LIN {X 0,Y 168.479,Z 365.357,A -85,B 0,C 180,E1 -26143.185,E2 -26143.185} C_VEL
LIN {X 0,Y 172.542,Z 376.389,A -85,B 0,C 180,E1 -26145.975,E2 -26145.975} C_VEL
LIN {X 0,Y 176.909,Z 386.851,A -85,B 0,C 180,E1 -26149.006,E2 -26149.006} C_VEL
LIN {X 0,Y 181.024,Z 395.329,A -85,B 0,C 180,E1 -26151.737,E2 -26151.737} C_VEL
LIN {X 0,Y 187.387,Z 405.901,A -85,B 0,C 180,E1 -26155.598,E2 -26155.598} C_VEL
LIN {X 0,Y 193.546,Z 414.105,A -85,B 0,C 180,E1 -26158.901,E2 -26158.901} C_VEL
LIN {X 0,Y 201.697,Z 422.811,A -85,B 0,C 180,E1 -26162.738,E2 -26162.738} C_VEL
LIN {X 0,Y 211.071,Z 430.45,A -85,B 0,C 180,E1 -26166.449,E2 -26166.449} C_VEL
LIN {X 0,Y 223.559,Z 438.19,A -85,B 0,C 180,E1 -26170.576,E2 -26170.576} C_VEL
LIN {X 0,Y 237.874,Z 444.989,A -85,B 0,C 180,E1 -26174.579,E2 -26174.579} C_VEL
LIN {X 0,Y 246.269,Z 448.506,A -85,B 0,C 180,E1 -26176.803,E2 -26176.803} C_VEL
LIN {X 0,Y 253.879,Z 451.483,A -85,B 0,C 180,E1 -26178.827,E2 -26178.827} C_VEL
LIN {X 0,Y 260.174,Z 454.048,A -85,B 0,C 180,E1 -26180.673,E2 -26180.673} C_VEL
LIN {X 0,Y 265.402,Z 456.155,A -85,B 0,C 180,E1 -26182.392,E2 -26182.392} C_VEL
LIN {X 0,Y 269.49,Z 457.837,A -85,B 0,C 180,E1 -26184.012,E2 -26184.012} C_VEL
LIN {X 0,Y 272.317,Z 459.137,A -85,B 0,C 180,E1 -26185.559,E2 -26185.559} C_VEL
LIN {X 0,Y 274.967,Z 460.059,A -85,B 0,C 180,E1 -26187.07,E2 -26187.07} C_VEL
LIN {X 0,Y 276.58,Z 460.609,A -85,B 0,C 180,E1 -26188.544,E2 -26188.544} C_VEL
LIN {X 0,Y 277.495,Z 460.786,A -85,B 0,C 180,E1 -26190,E2 -26190} C_VEL
LIN {X 0,Y 276.59,Z 460.609,A -85,B 0,C 180,E1 -26191.456,E2 -26191.456} C_VEL
LIN {X 0,Y 274.514,Z 459.922,A -85,B 0,C 180,E1 -26193.194,E2 -26193.194} C_VEL
LIN {X 0,Y 272.314,Z 459.137,A -85,B 0,C 180,E1 -26194.441,E2 -26194.441} C_VEL
LIN {X 0,Y 268.697,Z 457.523,A -85,B 0,C 180,E1 -26196.329,E2 -26196.329} C_VEL
LIN {X 0,Y 265.405,Z 456.155,A -85,B 0,C 180,E1 -26197.608,E2 -26197.608} C_VEL
LIN {X 0,Y 260.168,Z 454.048,A -85,B 0,C 180,E1 -26199.328,E2 -26199.328} C_VEL
LIN {X 0,Y 251.344,Z 450.491,A -85,B 0,C 180,E1 -26201.863,E2 -26201.863} C_VEL
LIN {X 0,Y 239.95,Z 445.859,A -85,B 0,C 180,E1 -26204.865,E2 -26204.865} C_VEL
LIN {X 0,Y 226.946,Z 439.906,A -85,B 0,C 180,E1 -26208.442,E2 -26208.442} C_VEL
LIN {X 0,Y 213.379,Z 432.019,A -85,B 0,C 180,E1 -26212.749,E2 -26212.749} C_VEL
LIN {X 0,Y 202.838,Z 423.881,A -85,B 0,C 180,E1 -26216.771,E2 -26216.771} C_VEL
LIN {X 0,Y 195.211,Z 416.062,A -85,B 0,C 180,E1 -26220.267,E2 -26220.267} C_VEL
LIN {X 0,Y 188.321,Z 407.27,A -85,B 0,C 180,E1 -26223.869,E2 -26223.869} C_VEL
LIN {X 0,Y 182.818,Z 398.65,A -85,B 0,C 180,E1 -26227.094,E2 -26227.094} C_VEL
LIN {X 0,Y 178.539,Z 390.449,A -85,B 0,C 180,E1 -26229.863,E2 -26229.863} C_VEL
LIN {X 0,Y 174.431,Z 381.231,A -85,B 0,C 180,E1 -26232.669,E2 -26232.669} C_VEL
LIN {X 0,Y 170.461,Z 371.172,A -85,B 0,C 180,E1 -26235.399,E2 -26235.399} C_VEL
LIN {X 0,Y 166.541,Z 359.972,A -85,B 0,C 180,E1 -26238.043,E2 -26238.043} C_VEL
LIN {X 0,Y 161.005,Z 344.099,A -85,B 0,C 180,E1 -26241.47,E2 -26241.47} C_VEL
LIN {X 0,Y 157.401,Z 335.249,A -85,B 0,C 180,E1 -26243.828,E2 -26243.828} C_VEL
LIN {X 0,Y 153.095,Z 326.286,A -85,B 0,C 180,E1 -26246.861,E2 -26246.861} C_VEL
LIN {X 0,Y 148.607,Z 318.02,A -85,B 0,C 180,E1 -26250.423,E2 -26250.423} C_VEL
LIN {X 0,Y 144.236,Z 310.858,A -85,B 0,C 180,E1 -26254.476,E2 -26254.476} C_VEL
LIN {X 0,Y 141.455,Z 306.781,A -85,B 0,C 180,E1 -26257.5,E2 -26257.5} C_VEL
LIN {X 0,Y 138.818,Z 302.887,A -85,B 0,C 180,E1 -26260.923,E2 -26260.923} C_VEL
LIN {X 0,Y 136.47,Z 299.576,A -85,B 0,C 180,E1 -26264.698,E2 -26264.698} C_VEL
LIN {X 0,Y 135.748,Z 298.305,A -85,B 0,C 180,E1 -26266.148,E2 -26266.148} C_VEL
LIN {X 0,Y 133.362,Z 295.448,A -85,B 0,C 180,E1 -26272.431,E2 -26272.431} C_VEL
LIN {X 0,Y 132.753,Z 293.551,A -85,B 0,C 180,E1 -26276.207,E2 -26276.207} C_VEL
LIN {X 0,Y 132.567,Z 292.935,A -85,B 0,C 180,E1 -26280.002,E2 -26280.002} C_VEL
LIN {X 0,Y 132.838,Z 293.86,A -85,B 0,C 180,E1 -26284.173,E2 -26284.173} C_VEL
LIN {X 0,Y 135.419,Z 298.099,A -85,B 0,C 180,E1 -26292.839,E2 -26292.839} C_VEL
LIN {X 0,Y 136.074,Z 298.699,A -85,B 0,C 180,E1 -26294.108,E2 -26294.108} C_VEL
LIN {X 0,Y 138.286,Z 302.315,A -85,B 0,C 180,E1 -26297.947,E2 -26297.947} C_VEL
LIN {X 0,Y 139.47,Z 303.8,A -85,B 0,C 180,E1 -26299.599,E2 -26299.599} C_VEL
LIN {X 0,Y 142.595,Z 308.443,A -85,B 0,C 180,E1 -26303.416,E2 -26303.416} C_VEL
LIN {X 0,Y 145.282,Z 312.654,A -85,B 0,C 180,E1 -26306.196,E2 -26306.196} C_VEL
LIN {X 0,Y 147.772,Z 316.823,A -85,B 0,C 180,E1 -26308.497,E2 -26308.497} C_VEL
LIN {X 0,Y 151.056,Z 324.304,A -85,B 0,C 180,E1 -26311.368,E2 -26311.368} C_VEL
LIN {X 0,Y 155.191,Z 335.226,A -85,B 0,C 180,E1 -26314.649,E2 -26314.649} C_VEL
LIN {X 0,Y 156.553,Z 339.736,A -85,B 0,C 180,E1 -26315.706,E2 -26315.706} C_VEL
LIN {X 0,Y 154.15,Z 367.569,A -85,B 0,C 180,E1 -26316.786,E2 -26316.786} C_VEL
LIN {X 0,Y 152.045,Z 380.407,A -85,B 0,C 180,E1 -26317.581,E2 -26317.581} C_VEL
LIN {X 0,Y 148.731,Z 393.184,A -85,B 0,C 180,E1 -26318.77,E2 -26318.77} C_VEL
LIN {X 0,Y 145.566,Z 402.693,A -85,B 0,C 180,E1 -26319.964,E2 -26319.964} C_VEL
LIN {X 0,Y 141.889,Z 411.963,A -85,B 0,C 180,E1 -26321.482,E2 -26321.482} C_VEL
LIN {X 0,Y 137.794,Z 420.904,A -85,B 0,C 180,E1 -26323.381,E2 -26323.381} C_VEL
LIN {X 0,Y 133.305,Z 429.426,A -85,B 0,C 180,E1 -26325.689,E2 -26325.689} C_VEL
LIN {X 0,Y 129.058,Z 436.64,A -85,B 0,C 180,E1 -26328.158,E2 -26328.158} C_VEL
LIN {X 0,Y 125.1,Z 442.839,A -85,B 0,C 180,E1 -26330.802,E2 -26330.802} C_VEL
LIN {X 0,Y 120.656,Z 449.376,A -85,B 0,C 180,E1 -26334.375,E2 -26334.375} C_VEL
LIN {X 0,Y 115.978,Z 455.795,A -85,B 0,C 180,E1 -26338.997,E2 -26338.997} C_VEL
LIN {X 0,Y 111.963,Z 460.925,A -85,B 0,C 180,E1 -26343.935,E2 -26343.935} C_VEL
LIN {X 0,Y 108.804,Z 464.915,A -85,B 0,C 180,E1 -26349.191,E2 -26349.191} C_VEL
LIN {X 0,Y 106.703,Z 467.874,A -85,B 0,C 180,E1 -26354.725,E2 -26354.725} C_VEL
LIN {X 0,Y 105.26,Z 470.336,A -85,B 0,C 180,E1 -26362.326,E2 -26362.326} C_VEL
LIN {X 0,Y 105.047,Z 470.932,A -85,B 0,C 180,E1 -26366.164,E2 -26366.164} C_VEL
LIN {X 0,Y 105.171,Z 471.094,A -85,B 0,C 180,E1 -26370,E2 -26370} C_VEL
LIN {X 0,Y 105.037,Z 470.932,A -85,B 0,C 180,E1 -26373.836,E2 -26373.836} C_VEL
LIN {X 0,Y 105.221,Z 470.335,A -85,B 0,C 180,E1 -26377.677,E2 -26377.677} C_VEL
LIN {X 0,Y 106.666,Z 467.873,A -85,B 0,C 180,E1 -26385.281,E2 -26385.281} C_VEL
LIN {X 0,Y 108.804,Z 464.915,A -85,B 0,C 180,E1 -26390.809,E2 -26390.809} C_VEL
LIN {X 0,Y 111.962,Z 460.925,A -85,B 0,C 180,E1 -26396.065,E2 -26396.065} C_VEL
LIN {X 0,Y 115.965,Z 455.795,A -85,B 0,C 180,E1 -26401.007,E2 -26401.007} C_VEL
LIN {X 0,Y 120.653,Z 449.376,A -85,B 0,C 180,E1 -26405.626,E2 -26405.626} C_VEL
LIN {X 0,Y 126.045,Z 441.455,A -85,B 0,C 180,E1 -26409.882,E2 -26409.882} C_VEL
LIN {X 0,Y 131.144,Z 433.262,A -85,B 0,C 180,E1 -26413.099,E2 -26413.099} C_VEL
LIN {X 0,Y 136.077,Z 424.305,A -85,B 0,C 180,E1 -26415.775,E2 -26415.775} C_VEL
LIN {X 0,Y 140.078,Z 416.014,A -85,B 0,C 180,E1 -26417.734,E2 -26417.734} C_VEL
LIN {X 0,Y 144.316,Z 405.955,A -85,B 0,C 180,E1 -26419.545,E2 -26419.545} C_VEL
LIN {X 0,Y 147.754,Z 396.202,A -85,B 0,C 180,E1 -26420.887,E2 -26420.887} C_VEL
LIN {X 0,Y 150.623,Z 386.126,A -85,B 0,C 180,E1 -26421.941,E2 -26421.941} C_VEL
LIN {X 0,Y 152.867,Z 375.717,A -85,B 0,C 180,E1 -26422.747,E2 -26422.747} C_VEL
LIN {X 0,Y 154.387,Z 365.529,A -85,B 0,C 180,E1 -26423.295,E2 -26423.295} C_VEL
LIN {X 0,Y 156.505,Z 339.441,A -85,B 0,C 180,E1 -26424.342,E2 -26424.342} C_VEL
LIN {X 0,Y 153.574,Z 330.813,A -85,B 0,C 180,E1 -26426.591,E2 -26426.591} C_VEL
LIN {X 0,Y 149.887,Z 321.54,A -85,B 0,C 180,E1 -26429.621,E2 -26429.621} C_VEL
LIN {X 0,Y 147.162,Z 315.702,A -85,B 0,C 180,E1 -26432.054,E2 -26432.054} C_VEL
LIN {X 0,Y 143.791,Z 310.303,A -85,B 0,C 180,E1 -26435.3,E2 -26435.3} C_VEL
LIN {X 0,Y 141.753,Z 307.117,A -85,B 0,C 180,E1 -26437.547,E2 -26437.547} C_VEL
LIN {X 0,Y 140.373,Z 306.364,A -85,B 0,C 180,E1 -26439.042,E2 -26439.042} C_VEL
LIN {X 0,Y 135.987,Z 307.211,A -85,B 0,C 180,E1 -26444.335,E2 -26444.335} C_VEL
LIN {X 0,Y 135.091,Z 306.305,A -85,B 0,C 180,E1 -26445.924,E2 -26445.924} C_VEL
LIN {X 0,Y 134.567,Z 305.22,A -85,B 0,C 180,E1 -26447.078,E2 -26447.078} C_VEL
LIN {X 0,Y 132.204,Z 301.989,A -85,B 0,C 180,E1 -26454.087,E2 -26454.087} C_VEL
LIN {X 0,Y 131.781,Z 300.34,A -85,B 0,C 180,E1 -26457.706,E2 -26457.706} C_VEL
LIN {X 0,Y 131.702,Z 299.984,A -85,B 0,C 180,E1 -26459.998,E2 -26459.998} C_VEL
LIN {X 0,Y 131.918,Z 300.847,A -85,B 0,C 180,E1 -26464.199,E2 -26464.199} C_VEL
LIN {X 0,Y 134.157,Z 304.913,A -85,B 0,C 180,E1 -26472.454,E2 -26472.454} C_VEL
LIN {X 0,Y 134.778,Z 305.568,A -85,B 0,C 180,E1 -26473.762,E2 -26473.762} C_VEL
LIN {X 0,Y 137.237,Z 309.489,A -85,B 0,C 180,E1 -26478.173,E2 -26478.173} C_VEL
LIN {X 0,Y 140.562,Z 314.653,A -85,B 0,C 180,E1 -26482.651,E2 -26482.651} C_VEL
LIN {X 0,Y 143.908,Z 320.11,A -85,B 0,C 180,E1 -26486.294,E2 -26486.294} C_VEL
LIN {X 0,Y 147.845,Z 327.198,A -85,B 0,C 180,E1 -26489.941,E2 -26489.941} C_VEL
LIN {X 0,Y 152.298,Z 336.274,A -85,B 0,C 180,E1 -26493.523,E2 -26493.523} C_VEL
LIN {X 0,Y 156.232,Z 345.744,A -85,B 0,C 180,E1 -26496.385,E2 -26496.385} C_VEL
LIN {X 0,Y 160.334,Z 358.02,A -85,B 0,C 180,E1 -26499.258,E2 -26499.258} C_VEL
LIN {X 0,Y 163.619,Z 368.614,A -85,B 0,C 180,E1 -26501.74,E2 -26501.74} C_VEL
LIN {X 0,Y 166.649,Z 377.879,A -85,B 0,C 180,E1 -26504.198,E2 -26504.198} C_VEL
LIN {X 0,Y 169.964,Z 386.802,A -85,B 0,C 180,E1 -26506.88,E2 -26506.88} C_VEL
LIN {X 0,Y 174.041,Z 396.438,A -85,B 0,C 180,E1 -26510.105,E2 -26510.105} C_VEL
LIN {X 0,Y 178.97,Z 405.713,A -85,B 0,C 180,E1 -26513.612,E2 -26513.612} C_VEL
LIN {X 0,Y 184.343,Z 413.859,A -85,B 0,C 180,E1 -26517.005,E2 -26517.005} C_VEL
LIN {X 0,Y 190.846,Z 421.669,A -85,B 0,C 180,E1 -26520.576,E2 -26520.576} C_VEL
LIN {X 0,Y 198.48,Z 428.958,A -85,B 0,C 180,E1 -26524.202,E2 -26524.202} C_VEL
LIN {X 0,Y 208.831,Z 436.357,A -85,B 0,C 180,E1 -26528.273,E2 -26528.273} C_VEL
LIN {X 0,Y 221.286,Z 443.055,A -85,B 0,C 180,E1 -26532.321,E2 -26532.321} C_VEL
LIN {X 0,Y 235.113,Z 448.819,A -85,B 0,C 180,E1 -26536.165,E2 -26536.165} C_VEL
LIN {X 0,Y 246.762,Z 453.049,A -85,B 0,C 180,E1 -26539.287,E2 -26539.287} C_VEL
LIN {X 0,Y 250.341,Z 454.315,A -85,B 0,C 180,E1 -26540.303,E2 -26540.303} C_VEL
LIN {X 0,Y 256.375,Z 456.402,A -85,B 0,C 180,E1 -26542.122,E2 -26542.122} C_VEL
LIN {X 0,Y 261.472,Z 458.211,A -85,B 0,C 180,E1 -26543.983,E2 -26543.983} C_VEL
LIN {X 0,Y 264.47,Z 459.349,A -85,B 0,C 180,E1 -26545.427,E2 -26545.427} C_VEL
LIN {X 0,Y 267.409,Z 460.312,A -85,B 0,C 180,E1 -26547.069,E2 -26547.069} C_VEL
LIN {X 0,Y 269.257,Z 460.807,A -85,B 0,C 180,E1 -26548.504,E2 -26548.504} C_VEL
LIN {X 0,Y 270.327,Z 460.977,A -85,B 0,C 180,E1 -26550,E2 -26550} C_VEL
LIN {X 0,Y 269.264,Z 460.807,A -85,B 0,C 180,E1 -26551.496,E2 -26551.496} C_VEL
LIN {X 0,Y 267.259,Z 460.27,A -85,B 0,C 180,E1 -26553.015,E2 -26553.015} C_VEL
LIN {X 0,Y 264.443,Z 459.349,A -85,B 0,C 180,E1 -26554.573,E2 -26554.573} C_VEL
LIN {X 0,Y 261.037,Z 458.069,A -85,B 0,C 180,E1 -26556.182,E2 -26556.182} C_VEL
LIN {X 0,Y 255.572,Z 456.138,A -85,B 0,C 180,E1 -26558.13,E2 -26558.13} C_VEL
LIN {X 0,Y 249.683,Z 454.083,A -85,B 0,C 180,E1 -26559.886,E2 -26559.886} C_VEL
LIN {X 0,Y 243.138,Z 451.778,A -85,B 0,C 180,E1 -26561.674,E2 -26561.674} C_VEL
LIN {X 0,Y 232.36,Z 447.741,A -85,B 0,C 180,E1 -26564.566,E2 -26564.566} C_VEL
LIN {X 0,Y 221.299,Z 443.027,A -85,B 0,C 180,E1 -26567.689,E2 -26567.689} C_VEL
LIN {X 0,Y 208.858,Z 436.356,A -85,B 0,C 180,E1 -26571.725,E2 -26571.725} C_VEL
LIN {X 0,Y 200.699,Z 430.75,A -85,B 0,C 180,E1 -26574.848,E2 -26574.848} C_VEL
LIN {X 0,Y 193.245,Z 424.166,A -85,B 0,C 180,E1 -26578.215,E2 -26578.215} C_VEL
LIN {X 0,Y 186.275,Z 416.336,A -85,B 0,C 180,E1 -26581.884,E2 -26581.884} C_VEL
LIN {X 0,Y 180.695,Z 408.562,A -85,B 0,C 180,E1 -26585.239,E2 -26585.239} C_VEL
LIN {X 0,Y 175.593,Z 399.762,A -85,B 0,C 180,E1 -26588.698,E2 -26588.698} C_VEL
LIN {X 0,Y 171.748,Z 391.161,A -85,B 0,C 180,E1 -26591.687,E2 -26591.687} C_VEL
LIN {X 0,Y 168.397,Z 382.706,A -85,B 0,C 180,E1 -26594.384,E2 -26594.384} C_VEL
LIN {X 0,Y 164.92,Z 372.651,A -85,B 0,C 180,E1 -26597.223,E2 -26597.223} C_VEL
LIN {X 0,Y 161.358,Z 361.267,A -85,B 0,C 180,E1 -26600.028,E2 -26600.028} C_VEL
LIN {X 0,Y 157.135,Z 348.285,A -85,B 0,C 180,E1 -26602.977,E2 -26602.977} C_VEL
LIN {X 0,Y 153.766,Z 339.696,A -85,B 0,C 180,E1 -26605.376,E2 -26605.376} C_VEL
LIN {X 0,Y 149.798,Z 331.089,A -85,B 0,C 180,E1 -26608.425,E2 -26608.425} C_VEL
LIN {X 0,Y 145.89,Z 323.573,A -85,B 0,C 180,E1 -26611.802,E2 -26611.802} C_VEL
LIN {X 0,Y 141.921,Z 316.824,A -85,B 0,C 180,E1 -26615.791,E2 -26615.791} C_VEL
LIN {X 0,Y 139.553,Z 313.107,A -85,B 0,C 180,E1 -26618.587,E2 -26618.587} C_VEL
LIN {X 0,Y 137.239,Z 309.488,A -85,B 0,C 180,E1 -26621.826,E2 -26621.826} C_VEL
LIN {X 0,Y 134.859,Z 305.757,A -85,B 0,C 180,E1 -26626.055,E2 -26626.055} C_VEL
LIN {X 0,Y 134.162,Z 304.871,A -85,B 0,C 180,E1 -26627.546,E2 -26627.546} C_VEL
LIN {X 0,Y 132.174,Z 301.855,A -85,B 0,C 180,E1 -26633.897,E2 -26633.897} C_VEL
LIN {X 0,Y 131.811,Z 300.43,A -85,B 0,C 180,E1 -26636.945,E2 -26636.945} C_VEL
LIN {X 0,Y 131.707,Z 300.081,A -85,B 0,C 180,E1 -26640.766,E2 -26640.766} C_VEL
LIN {X 0,Y 131.925,Z 300.918,A -85,B 0,C 180,E1 -26643.915,E2 -26643.915} C_VEL
LIN {X 0,Y 134.298,Z 305.023,A -85,B 0,C 180,E1 -26652.372,E2 -26652.372} C_VEL
LIN {X 0,Y 134.859,Z 305.768,A -85,B 0,C 180,E1 -26653.565,E2 -26653.565} C_VEL
LIN {X 0,Y 137.95,Z 310.612,A -85,B 0,C 180,E1 -26658.858,E2 -26658.858} C_VEL
LIN {X 0,Y 140.594,Z 314.65,A -85,B 0,C 180,E1 -26662.3,E2 -26662.3} C_VEL
LIN {X 0,Y 144.211,Z 320.604,A -85,B 0,C 180,E1 -26666.211,E2 -26666.211} C_VEL
LIN {X 0,Y 146.759,Z 326.225,A -85,B 0,C 180,E1 -26668.712,E2 -26668.712} C_VEL
LIN {X 0,Y 150.274,Z 335.658,A -85,B 0,C 180,E1 -26671.894,E2 -26671.894} C_VEL
LIN {X 0,Y 152.306,Z 342.009,A -85,B 0,C 180,E1 -26673.625,E2 -26673.625} C_VEL
LIN {X 0,Y 150.039,Z 367.082,A -85,B 0,C 180,E1 -26674.597,E2 -26674.597} C_VEL
LIN {X 0,Y 147.79,Z 380.354,A -85,B 0,C 180,E1 -26675.408,E2 -26675.408} C_VEL
LIN {X 0,Y 144.398,Z 392.992,A -85,B 0,C 180,E1 -26676.576,E2 -26676.576} C_VEL
LIN {X 0,Y 141.112,Z 402.501,A -85,B 0,C 180,E1 -26677.755,E2 -26677.755} C_VEL
LIN {X 0,Y 137.277,Z 411.77,A -85,B 0,C 180,E1 -26679.256,E2 -26679.256} C_VEL
LIN {X 0,Y 133.008,Z 420.711,A -85,B 0,C 180,E1 -26681.153,E2 -26681.153} C_VEL
LIN {X 0,Y 128.322,Z 429.234,A -85,B 0,C 180,E1 -26683.475,E2 -26683.475} C_VEL
LIN {X 0,Y 123.832,Z 436.447,A -85,B 0,C 180,E1 -26685.954,E2 -26685.954} C_VEL
LIN {X 0,Y 119.662,Z 442.645,A -85,B 0,C 180,E1 -26688.644,E2 -26688.644} C_VEL
LIN {X 0,Y 114.934,Z 449.182,A -85,B 0,C 180,E1 -26692.304,E2 -26692.304} C_VEL
LIN {X 0,Y 111.518,Z 453.685,A -85,B 0,C 180,E1 -26695.446,E2 -26695.446} C_VEL
LIN {X 0,Y 106.899,Z 459.176,A -85,B 0,C 180,E1 -26700.457,E2 -26700.457} C_VEL
LIN {X 0,Y 103.208,Z 463.503,A -85,B 0,C 180,E1 -26705.885,E2 -26705.885} C_VEL
LIN {X 0,Y 101.256,Z 465.874,A -85,B 0,C 180,E1 -26709.694,E2 -26709.694} C_VEL
LIN {X 0,Y 99.828,Z 467.68,A -85,B 0,C 180,E1 -26713.644,E2 -26713.644} C_VEL
LIN {X 0,Y 98.209,Z 470.142,A -85,B 0,C 180,E1 -26721.771,E2 -26721.771} C_VEL
LIN {X 0,Y 97.952,Z 470.739,A -85,B 0,C 180,E1 -26725.886,E2 -26725.886} C_VEL
LIN {X 0,Y 98.077,Z 470.902,A -85,B 0,C 180,E1 -26730,E2 -26730} C_VEL
LIN {X 0,Y 97.943,Z 470.739,A -85,B 0,C 180,E1 -26734.115,E2 -26734.115} C_VEL
LIN {X 0,Y 98.178,Z 470.141,A -85,B 0,C 180,E1 -26738.231,E2 -26738.231} C_VEL
LIN {X 0,Y 99.798,Z 467.679,A -85,B 0,C 180,E1 -26746.361,E2 -26746.361} C_VEL
LIN {X 0,Y 102.181,Z 464.722,A -85,B 0,C 180,E1 -26752.228,E2 -26752.228} C_VEL
LIN {X 0,Y 105.595,Z 460.731,A -85,B 0,C 180,E1 -26757.768,E2 -26757.768} C_VEL
LIN {X 0,Y 109.929,Z 455.602,A -85,B 0,C 180,E1 -26762.917,E2 -26762.917} C_VEL
LIN {X 0,Y 114.092,Z 450.286,A -85,B 0,C 180,E1 -26766.962,E2 -26766.962} C_VEL
LIN {X 0,Y 118.658,Z 444.02,A -85,B 0,C 180,E1 -26770.656,E2 -26770.656} C_VEL
LIN {X 0,Y 122.787,Z 438.073,A -85,B 0,C 180,E1 -26773.381,E2 -26773.381} C_VEL
LIN {X 0,Y 127.157,Z 431.15,A -85,B 0,C 180,E1 -26775.931,E2 -26775.931} C_VEL
LIN {X 0,Y 131.807,Z 422.978,A -85,B 0,C 180,E1 -26778.287,E2 -26778.287} C_VEL
LIN {X 0,Y 136.035,Z 414.471,A -85,B 0,C 180,E1 -26780.218,E2 -26780.218} C_VEL
LIN {X 0,Y 139.808,Z 405.762,A -85,B 0,C 180,E1 -26781.762,E2 -26781.762} C_VEL
LIN {X 0,Y 143.391,Z 396.01,A -85,B 0,C 180,E1 -26783.084,E2 -26783.084} C_VEL
LIN {X 0,Y 146.359,Z 385.933,A -85,B 0,C 180,E1 -26784.127,E2 -26784.127} C_VEL
LIN {X 0,Y 148.53,Z 376.276,A -85,B 0,C 180,E1 -26784.879,E2 -26784.879} C_VEL
LIN {X 0,Y 150.171,Z 366.091,A -85,B 0,C 180,E1 -26785.427,E2 -26785.427} C_VEL
LIN {X 0,Y 152.308,Z 341.993,A -85,B 0,C 180,E1 -26786.376,E2 -26786.376} C_VEL
LIN {X 0,Y 149.957,Z 334.8,A -85,B 0,C 180,E1 -26788.376,E2 -26788.376} C_VEL
LIN {X 0,Y 146.839,Z 326.47,A -85,B 0,C 180,E1 -26791.208,E2 -26791.208} C_VEL
LIN {X 0,Y 144.294,Z 320.735,A -85,B 0,C 180,E1 -26793.708,E2 -26793.708} C_VEL
LIN {X 0,Y 140.107,Z 313.769,A -85,B 0,C 180,E1 -26798.304,E2 -26798.304} C_VEL
LIN {X 0,Y 137.065,Z 309.285,A -85,B 0,C 180,E1 -26802.466,E2 -26802.466} C_VEL
LIN {X 0,Y 135.091,Z 306.305,A -85,B 0,C 180,E1 -26805.924,E2 -26805.924} C_VEL
LIN {X 0,Y 134.359,Z 305.169,A -85,B 0,C 180,E1 -26807.476,E2 -26807.476} C_VEL
LIN {X 0,Y 133.244,Z 304.74,A -85,B 0,C 180,E1 -26809.939,E2 -26809.939} C_VEL
LIN {X 0,Y 131.692,Z 305.939,A -85,B 0,C 180,E1 -26814.187,E2 -26814.187} C_VEL
LIN {X 0,Y 130.877,Z 307.119,A -85,B 0,C 180,E1 -26818.579,E2 -26818.579} C_VEL
LIN {X 0,Y 130.838,Z 307.095,A -85,B 0,C 180,E1 -26819.468,E2 -26819.468} C_VEL
LIN {X 0,Y 130.969,Z 307.678,A -85,B 0,C 180,E1 -26823.459,E2 -26823.459} C_VEL
LIN {X 0,Y 132.983,Z 311.787,A -85,B 0,C 180,E1 -26831.824,E2 -26831.824} C_VEL
LIN {X 0,Y 133.57,Z 312.561,A -85,B 0,C 180,E1 -26833.171,E2 -26833.171} C_VEL
LIN {X 0,Y 136.341,Z 317.175,A -85,B 0,C 180,E1 -26838.297,E2 -26838.297} C_VEL
LIN {X 0,Y 138.859,Z 321.337,A -85,B 0,C 180,E1 -26841.823,E2 -26841.823} C_VEL
LIN {X 0,Y 141.692,Z 326.216,A -85,B 0,C 180,E1 -26845.13,E2 -26845.13} C_VEL
LIN {X 0,Y 145.284,Z 333.104,A -85,B 0,C 180,E1 -26848.727,E2 -26848.727} C_VEL
LIN {X 0,Y 149.381,Z 342.043,A -85,B 0,C 180,E1 -26852.296,E2 -26852.296} C_VEL
LIN {X 0,Y 152.673,Z 350.479,A -85,B 0,C 180,E1 -26854.903,E2 -26854.903} C_VEL
LIN {X 0,Y 156.081,Z 361.51,A -85,B 0,C 180,E1 -26857.638,E2 -26857.638} C_VEL
LIN {X 0,Y 158.454,Z 370.323,A -85,B 0,C 180,E1 -26859.816,E2 -26859.816} C_VEL
LIN {X 0,Y 160.646,Z 378.117,A -85,B 0,C 180,E1 -26861.951,E2 -26861.951} C_VEL
LIN {X 0,Y 163.869,Z 388.405,A -85,B 0,C 180,E1 -26865.151,E2 -26865.151} C_VEL
LIN {X 0,Y 167.12,Z 397.069,A -85,B 0,C 180,E1 -26868.19,E2 -26868.19} C_VEL
LIN {X 0,Y 170.834,Z 405.401,A -85,B 0,C 180,E1 -26871.409,E2 -26871.409} C_VEL
LIN {X 0,Y 176.395,Z 414.906,A -85,B 0,C 180,E1 -26875.559,E2 -26875.559} C_VEL
LIN {X 0,Y 181.738,Z 421.97,A -85,B 0,C 180,E1 -26878.951,E2 -26878.951} C_VEL
LIN {X 0,Y 189.22,Z 429.789,A -85,B 0,C 180,E1 -26883.048,E2 -26883.048} C_VEL
LIN {X 0,Y 198.337,Z 436.791,A -85,B 0,C 180,E1 -26887.114,E2 -26887.114} C_VEL
LIN {X 0,Y 208.358,Z 442.584,A -85,B 0,C 180,E1 -26890.809,E2 -26890.809} C_VEL
LIN {X 0,Y 219.136,Z 447.41,A -85,B 0,C 180,E1 -26894.18,E2 -26894.18} C_VEL
LIN {X 0,Y 232.085,Z 452.082,A -85,B 0,C 180,E1 -26897.762,E2 -26897.762} C_VEL
LIN {X 0,Y 242.26,Z 455.294,A -85,B 0,C 180,E1 -26900.514,E2 -26900.514} C_VEL
LIN {X 0,Y 248.225,Z 457.108,A -85,B 0,C 180,E1 -26902.28,E2 -26902.28} C_VEL
LIN {X 0,Y 254.243,Z 458.919,A -85,B 0,C 180,E1 -26904.339,E2 -26904.339} C_VEL
LIN {X 0,Y 256.387,Z 459.567,A -85,B 0,C 180,E1 -26905.283,E2 -26905.283} C_VEL
LIN {X 0,Y 260.309,Z 460.676,A -85,B 0,C 180,E1 -26907.354,E2 -26907.354} C_VEL
LIN {X 0,Y 261.833,Z 461.008,A -85,B 0,C 180,E1 -26908.462,E2 -26908.462} C_VEL
LIN {X 0,Y 263.136,Z 461.168,A -85,B 0,C 180,E1 -26910,E2 -26910} C_VEL
LIN {X 0,Y 261.838,Z 461.007,A -85,B 0,C 180,E1 -26911.538,E2 -26911.538} C_VEL
LIN {X 0,Y 259.49,Z 460.482,A -85,B 0,C 180,E1 -26913.105,E2 -26913.105} C_VEL
LIN {X 0,Y 256.372,Z 459.567,A -85,B 0,C 180,E1 -26914.717,E2 -26914.717} C_VEL
LIN {X 0,Y 254.243,Z 458.92,A -85,B 0,C 180,E1 -26915.66,E2 -26915.66} C_VEL
LIN {X 0,Y 248.225,Z 457.108,A -85,B 0,C 180,E1 -26917.72,E2 -26917.72} C_VEL
LIN {X 0,Y 239.922,Z 454.596,A -85,B 0,C 180,E1 -26920.123,E2 -26920.123} C_VEL
LIN {X 0,Y 230.494,Z 451.563,A -85,B 0,C 180,E1 -26922.658,E2 -26922.658} C_VEL
LIN {X 0,Y 219.14,Z 447.401,A -85,B 0,C 180,E1 -26925.824,E2 -26925.824} C_VEL
LIN {X 0,Y 206.255,Z 441.488,A -85,B 0,C 180,E1 -26929.922,E2 -26929.922} C_VEL
LIN {X 0,Y 196.267,Z 435.387,A -85,B 0,C 180,E1 -26933.748,E2 -26933.748} C_VEL
LIN {X 0,Y 187.142,Z 427.784,A -85,B 0,C 180,E1 -26938.054,E2 -26938.054} C_VEL
LIN {X 0,Y 179.291,Z 418.917,A -85,B 0,C 180,E1 -26942.57,E2 -26942.57} C_VEL
LIN {X 0,Y 173.202,Z 409.793,A -85,B 0,C 180,E1 -26946.74,E2 -26946.74} C_VEL
LIN {X 0,Y 169.134,Z 401.905,A -85,B 0,C 180,E1 -26950.007,E2 -26950.007} C_VEL
LIN {X 0,Y 165.129,Z 391.922,A -85,B 0,C 180,E1 -26953.655,E2 -26953.655} C_VEL
LIN {X 0,Y 162.036,Z 382.699,A -85,B 0,C 180,E1 -26956.674,E2 -26956.674} C_VEL
LIN {X 0,Y 158.946,Z 372.137,A -85,B 0,C 180,E1 -26959.712,E2 -26959.712} C_VEL
LIN {X 0,Y 155.937,Z 360.94,A -85,B 0,C 180,E1 -26962.525,E2 -26962.525} C_VEL
LIN {X 0,Y 152.677,Z 350.493,A -85,B 0,C 180,E1 -26965.094,E2 -26965.094} C_VEL
LIN {X 0,Y 149.475,Z 342.254,A -85,B 0,C 180,E1 -26967.628,E2 -26967.628} C_VEL
LIN {X 0,Y 145.285,Z 333.096,A -85,B 0,C 180,E1 -26971.273,E2 -26971.273} C_VEL
LIN {X 0,Y 141.69,Z 326.232,A -85,B 0,C 180,E1 -26974.87,E2 -26974.87} C_VEL
LIN {X 0,Y 139.196,Z 321.927,A -85,B 0,C 180,E1 -26977.75,E2 -26977.75} C_VEL
LIN {X 0,Y 137.53,Z 319.166,A -85,B 0,C 180,E1 -26979.944,E2 -26979.944} C_VEL
LIN {X 0,Y 135.568,Z 315.944,A -85,B 0,C 180,E1 -26982.95,E2 -26982.95} C_VEL
LIN {X 0,Y 133.307,Z 312.004,A -85,B 0,C 180,E1 -26987.465,E2 -26987.465} C_VEL
LIN {X 0,Y 131.241,Z 308.956,A -85,B 0,C 180,E1 -26994.143,E2 -26994.143} C_VEL
LIN {X 0,Y 130.94,Z 307.531,A -85,B 0,C 180,E1 -26996.925,E2 -26996.925} C_VEL
LIN {X 0,Y 130.842,Z 307.127,A -85,B 0,C 180,E1 -27000.771,E2 -27000.771} C_VEL
LIN {X 0,Y 131.049,Z 308.068,A -85,B 0,C 180,E1 -27003.942,E2 -27003.942} C_VEL
LIN {X 0,Y 133.112,Z 311.88,A -85,B 0,C 180,E1 -27011.732,E2 -27011.732} C_VEL
LIN {X 0,Y 133.622,Z 312.703,A -85,B 0,C 180,E1 -27012.918,E2 -27012.918} C_VEL
LIN {X 0,Y 136.289,Z 317.073,A -85,B 0,C 180,E1 -27017.831,E2 -27017.831} C_VEL
LIN {X 0,Y 138.782,Z 321.164,A -85,B 0,C 180,E1 -27021.337,E2 -27021.337} C_VEL
LIN {X 0,Y 141.981,Z 326.752,A -85,B 0,C 180,E1 -27025.06,E2 -27025.06} C_VEL
LIN {X 0,Y 144.559,Z 333.019,A -85,B 0,C 180,E1 -27027.804,E2 -27027.804} C_VEL
LIN {X 0,Y 148.18,Z 343.951,A -85,B 0,C 180,E1 -27031.34,E2 -27031.34} C_VEL
LIN {X 0,Y 148.118,Z 346.245,A -85,B 0,C 180,E1 -27031.508,E2 -27031.508} C_VEL
LIN {X 0,Y 146.034,Z 367.636,A -85,B 0,C 180,E1 -27032.343,E2 -27032.343} C_VEL
LIN {X 0,Y 143.414,Z 381.697,A -85,B 0,C 180,E1 -27033.22,E2 -27033.22} C_VEL
LIN {X 0,Y 140.285,Z 392.799,A -85,B 0,C 180,E1 -27034.248,E2 -27034.248} C_VEL
LIN {X 0,Y 136.878,Z 402.308,A -85,B 0,C 180,E1 -27035.403,E2 -27035.403} C_VEL
LIN {X 0,Y 132.907,Z 411.578,A -85,B 0,C 180,E1 -27036.89,E2 -27036.89} C_VEL
LIN {X 0,Y 128.432,Z 420.517,A -85,B 0,C 180,E1 -27038.76,E2 -27038.76} C_VEL
LIN {X 0,Y 123.546,Z 429.041,A -85,B 0,C 180,E1 -27041.085,E2 -27041.085} C_VEL
LIN {X 0,Y 118.817,Z 436.253,A -85,B 0,C 180,E1 -27043.566,E2 -27043.566} C_VEL
LIN {X 0,Y 114.399,Z 442.451,A -85,B 0,C 180,E1 -27046.28,E2 -27046.28} C_VEL
LIN {X 0,Y 109.365,Z 448.988,A -85,B 0,C 180,E1 -27050.013,E2 -27050.013} C_VEL
LIN {X 0,Y 104.016,Z 455.408,A -85,B 0,C 180,E1 -27054.948,E2 -27054.948} C_VEL
LIN {X 0,Y 99.324,Z 460.537,A -85,B 0,C 180,E1 -27060.31,E2 -27060.31} C_VEL
LIN {X 0,Y 95.608,Z 464.528,A -85,B 0,C 180,E1 -27066.153,E2 -27066.153} C_VEL
LIN {X 0,Y 93.003,Z 467.486,A -85,B 0,C 180,E1 -27072.406,E2 -27072.406} C_VEL
LIN {X 0,Y 91.164,Z 469.949,A -85,B 0,C 180,E1 -27081.131,E2 -27081.131} C_VEL
LIN {X 0,Y 90.88,Z 470.547,A -85,B 0,C 180,E1 -27085.565,E2 -27085.565} C_VEL
LIN {X 0,Y 90.976,Z 470.709,A -85,B 0,C 180,E1 -27090,E2 -27090} C_VEL
LIN {X 0,Y 90.873,Z 470.546,A -85,B 0,C 180,E1 -27094.436,E2 -27094.436} C_VEL
LIN {X 0,Y 91.138,Z 469.948,A -85,B 0,C 180,E1 -27098.872,E2 -27098.872} C_VEL
LIN {X 0,Y 92.979,Z 467.486,A -85,B 0,C 180,E1 -27107.599,E2 -27107.599} C_VEL
LIN {X 0,Y 95.608,Z 464.528,A -85,B 0,C 180,E1 -27113.847,E2 -27113.847} C_VEL
LIN {X 0,Y 99.322,Z 460.537,A -85,B 0,C 180,E1 -27119.69,E2 -27119.69} C_VEL
LIN {X 0,Y 104.008,Z 455.408,A -85,B 0,C 180,E1 -27125.055,E2 -27125.055} C_VEL
LIN {X 0,Y 109.36,Z 448.988,A -85,B 0,C 180,E1 -27129.989,E2 -27129.989} C_VEL
LIN {X 0,Y 115.494,Z 441.069,A -85,B 0,C 180,E1 -27134.41,E2 -27134.41} C_VEL
LIN {X 0,Y 121.144,Z 432.875,A -85,B 0,C 180,E1 -27137.703,E2 -27137.703} C_VEL
LIN {X 0,Y 126.576,Z 423.919,A -85,B 0,C 180,E1 -27140.389,E2 -27140.389} C_VEL
LIN {X 0,Y 130.951,Z 415.628,A -85,B 0,C 180,E1 -27142.336,E2 -27142.336} C_VEL
LIN {X 0,Y 135.533,Z 405.569,A -85,B 0,C 180,E1 -27144.118,E2 -27144.118} C_VEL
LIN {X 0,Y 139.25,Z 395.818,A -85,B 0,C 180,E1 -27145.416,E2 -27145.416} C_VEL
LIN {X 0,Y 142.316,Z 385.74,A -85,B 0,C 180,E1 -27146.443,E2 -27146.443} C_VEL
LIN {X 0,Y 144.682,Z 375.482,A -85,B 0,C 180,E1 -27147.218,E2 -27147.218} C_VEL
LIN {X 0,Y 146.319,Z 365.419,A -85,B 0,C 180,E1 -27147.738,E2 -27147.738} C_VEL
LIN {X 0,Y 148.264,Z 344.353,A -85,B 0,C 180,E1 -27148.571,E2 -27148.571} C_VEL
LIN {X 0,Y 146.173,Z 337.686,A -85,B 0,C 180,E1 -27150.571,E2 -27150.571} C_VEL
LIN {X 0,Y 143.3,Z 329.775,A -85,B 0,C 180,E1 -27153.511,E2 -27153.511} C_VEL
LIN {X 0,Y 141.519,Z 325.961,A -85,B 0,C 180,E1 -27155.433,E2 -27155.433} C_VEL
LIN {X 0,Y 138.134,Z 319.987,A -85,B 0,C 180,E1 -27159.524,E2 -27159.524} C_VEL
LIN {X 0,Y 135.513,Z 315.851,A -85,B 0,C 180,E1 -27163.425,E2 -27163.425} C_VEL
LIN {X 0,Y 133.311,Z 312.06,A -85,B 0,C 180,E1 -27167.825,E2 -27167.825} C_VEL
LIN {X 0,Y 131.121,Z 308.457,A -85,B 0,C 180,E1 -27175.387,E2 -27175.387} C_VEL
LIN {X 0,Y 130.868,Z 307.256,A -85,B 0,C 180,E1 -27178.46,E2 -27178.46} C_VEL
LIN {X 0,Y 130.838,Z 307.095,A -85,B 0,C 180,E1 -27179.468,E2 -27179.468} C_VEL
LIN {X 0,Y 130.817,Z 307.339,A -85,B 0,C 180,E1 -27181.17,E2 -27181.17} C_VEL
LIN {X 0,Y 130.84,Z 308.932,A -85,B 0,C 180,E1 -27183.647,E2 -27183.647} C_VEL
LIN {X 0,Y 130.964,Z 311.456,A -85,B 0,C 180,E1 -27185.994,E2 -27185.994} C_VEL
LIN {X 0,Y 131.373,Z 315.507,A -85,B 0,C 180,E1 -27189.08,E2 -27189.08} C_VEL
LIN {X 0,Y 132.245,Z 319.17,A -85,B 0,C 180,E1 -27192.212,E2 -27192.212} C_VEL
LIN {X 0,Y 134.676,Z 323.541,A -85,B 0,C 180,E1 -27197.166,E2 -27197.166} C_VEL
LIN {X 0,Y 137.086,Z 327.797,A -85,B 0,C 180,E1 -27200.832,E2 -27200.832} C_VEL
LIN {X 0,Y 139.853,Z 332.901,A -85,B 0,C 180,E1 -27204.294,E2 -27204.294} C_VEL
LIN {X 0,Y 143.216,Z 339.893,A -85,B 0,C 180,E1 -27207.892,E2 -27207.892} C_VEL
LIN {X 0,Y 146.733,Z 348.236,A -85,B 0,C 180,E1 -27211.19,E2 -27211.19} C_VEL
LIN {X 0,Y 149.632,Z 356.394,A -85,B 0,C 180,E1 -27213.696,E2 -27213.696} C_VEL
LIN {X 0,Y 152.716,Z 368.599,A -85,B 0,C 180,E1 -27216.846,E2 -27216.846} C_VEL
LIN {X 0,Y 154.973,Z 378.353,A -85,B 0,C 180,E1 -27219.561,E2 -27219.561} C_VEL
LIN {X 0,Y 157.411,Z 387.674,A -85,B 0,C 180,E1 -27222.529,E2 -27222.529} C_VEL
LIN {X 0,Y 160.148,Z 396.684,A -85,B 0,C 180,E1 -27225.744,E2 -27225.744} C_VEL
LIN {X 0,Y 163.25,Z 405.125,A -85,B 0,C 180,E1 -27229.089,E2 -27229.089} C_VEL
LIN {X 0,Y 167.395,Z 413.685,A -85,B 0,C 180,E1 -27232.909,E2 -27232.909} C_VEL
LIN {X 0,Y 172.963,Z 422.274,A -85,B 0,C 180,E1 -27237.197,E2 -27237.197} C_VEL
LIN {X 0,Y 179.25,Z 429.579,A -85,B 0,C 180,E1 -27241.212,E2 -27241.212} C_VEL
LIN {X 0,Y 186.214,Z 435.779,A -85,B 0,C 180,E1 -27244.928,E2 -27244.928} C_VEL
LIN {X 0,Y 195.652,Z 442.008,A -85,B 0,C 180,E1 -27249.054,E2 -27249.054} C_VEL
LIN {X 0,Y 206.022,Z 447.095,A -85,B 0,C 180,E1 -27252.773,E2 -27252.773} C_VEL
LIN {X 0,Y 217.148,Z 451.293,A -85,B 0,C 180,E1 -27256.151,E2 -27256.151} C_VEL
LIN {X 0,Y 228.898,Z 454.894,A -85,B 0,C 180,E1 -27259.384,E2 -27259.384} C_VEL
LIN {X 0,Y 236.597,Z 456.944,A -85,B 0,C 180,E1 -27261.459,E2 -27261.459} C_VEL
LIN {X 0,Y 242.953,Z 458.565,A -85,B 0,C 180,E1 -27263.355,E2 -27263.355} C_VEL
LIN {X 0,Y 248.084,Z 459.791,A -85,B 0,C 180,E1 -27265.125,E2 -27265.125} C_VEL
LIN {X 0,Y 253.216,Z 460.999,A -85,B 0,C 180,E1 -27267.652,E2 -27267.652} C_VEL
LIN {X 0,Y 254.342,Z 461.21,A -85,B 0,C 180,E1 -27268.417,E2 -27268.417} C_VEL
LIN {X 0,Y 255.912,Z 461.36,A -85,B 0,C 180,E1 -27270,E2 -27270} C_VEL
LIN {X 0,Y 254.343,Z 461.21,A -85,B 0,C 180,E1 -27271.583,E2 -27271.583} C_VEL
LIN {X 0,Y 251.561,Z 460.699,A -85,B 0,C 180,E1 -27273.203,E2 -27273.203} C_VEL
LIN {X 0,Y 248.081,Z 459.791,A -85,B 0,C 180,E1 -27274.875,E2 -27274.875} C_VEL
LIN {X 0,Y 242.953,Z 458.566,A -85,B 0,C 180,E1 -27276.645,E2 -27276.645} C_VEL
LIN {X 0,Y 234.823,Z 456.495,A -85,B 0,C 180,E1 -27279.019,E2 -27279.019} C_VEL
LIN {X 0,Y 222.922,Z 453.174,A -85,B 0,C 180,E1 -27282.229,E2 -27282.229} C_VEL
LIN {X 0,Y 208.739,Z 448.215,A -85,B 0,C 180,E1 -27286.354,E2 -27286.354} C_VEL
LIN {X 0,Y 198.172,Z 443.361,A -85,B 0,C 180,E1 -27289.985,E2 -27289.985} C_VEL
LIN {X 0,Y 189.304,Z 438.014,A -85,B 0,C 180,E1 -27293.631,E2 -27293.631} C_VEL
LIN {X 0,Y 181.895,Z 432.138,A -85,B 0,C 180,E1 -27297.297,E2 -27297.297} C_VEL
LIN {X 0,Y 174.888,Z 424.723,A -85,B 0,C 180,E1 -27301.494,E2 -27301.494} C_VEL
LIN {X 0,Y 169.27,Z 416.872,A -85,B 0,C 180,E1 -27305.54,E2 -27305.54} C_VEL
LIN {X 0,Y 165.146,Z 409.409,A -85,B 0,C 180,E1 -27309.047,E2 -27309.047} C_VEL
LIN {X 0,Y 161.799,Z 401.466,A -85,B 0,C 180,E1 -27312.405,E2 -27312.405} C_VEL
LIN {X 0,Y 158.519,Z 391.655,A -85,B 0,C 180,E1 -27316.1,E2 -27316.1} C_VEL
LIN {X 0,Y 155.966,Z 382.361,A -85,B 0,C 180,E1 -27319.206,E2 -27319.206} C_VEL
LIN {X 0,Y 153.481,Z 372.03,A -85,B 0,C 180,E1 -27322.235,E2 -27322.235} C_VEL
LIN {X 0,Y 150.843,Z 360.544,A -85,B 0,C 180,E1 -27325.2,E2 -27325.2} C_VEL
LIN {X 0,Y 147.644,Z 350.591,A -85,B 0,C 180,E1 -27328.013,E2 -27328.013} C_VEL
LIN {X 0,Y 144.088,Z 341.908,A -85,B 0,C 180,E1 -27331.247,E2 -27331.247} C_VEL
LIN {X 0,Y 140.865,Z 334.927,A -85,B 0,C 180,E1 -27334.564,E2 -27334.564} C_VEL
LIN {X 0,Y 137.548,Z 328.66,A -85,B 0,C 180,E1 -27338.541,E2 -27338.541} C_VEL
LIN {X 0,Y 135.863,Z 325.665,A -85,B 0,C 180,E1 -27340.921,E2 -27340.921} C_VEL
LIN {X 0,Y 134.002,Z 322.429,A -85,B 0,C 180,E1 -27344.019,E2 -27344.019} C_VEL
LIN {X 0,Y 131.979,Z 318.719,A -85,B 0,C 180,E1 -27348.465,E2 -27348.465} C_VEL
LIN {X 0,Y 130.244,Z 315.784,A -85,B 0,C 180,E1 -27354.874,E2 -27354.874} C_VEL
LIN {X 0,Y 130.016,Z 314.437,A -85,B 0,C 180,E1 -27357.678,E2 -27357.678} C_VEL
LIN {X 0,Y 129.977,Z 314.175,A -85,B 0,C 180,E1 -27360.776,E2 -27360.776} C_VEL
LIN {X 0,Y 130.148,Z 315.296,A -85,B 0,C 180,E1 -27363.872,E2 -27363.872} C_VEL
LIN {X 0,Y 132.282,Z 319.3,A -85,B 0,C 180,E1 -27371.938,E2 -27371.938} C_VEL
LIN {X 0,Y 134.739,Z 323.646,A -85,B 0,C 180,E1 -27376.89,E2 -27376.89} C_VEL
LIN {X 0,Y 137.081,Z 327.791,A -85,B 0,C 180,E1 -27380.444,E2 -27380.444} C_VEL
LIN {X 0,Y 139.91,Z 333.121,A -85,B 0,C 180,E1 -27383.991,E2 -27383.991} C_VEL
LIN {X 0,Y 142.264,Z 339.664,A -85,B 0,C 180,E1 -27386.746,E2 -27386.746} C_VEL
LIN {X 0,Y 144.444,Z 346.766,A -85,B 0,C 180,E1 -27389.116,E2 -27389.116} C_VEL
LIN {X 0,Y 142.323,Z 367.728,A -85,B 0,C 180,E1 -27389.941,E2 -27389.941} C_VEL
LIN {X 0,Y 139.765,Z 381.081,A -85,B 0,C 180,E1 -27390.746,E2 -27390.746} C_VEL
LIN {X 0,Y 136.419,Z 392.606,A -85,B 0,C 180,E1 -27391.784,E2 -27391.784} C_VEL
LIN {X 0,Y 132.896,Z 402.115,A -85,B 0,C 180,E1 -27392.91,E2 -27392.91} C_VEL
LIN {X 0,Y 128.763,Z 411.385,A -85,B 0,C 180,E1 -27394.357,E2 -27394.357} C_VEL
LIN {X 0,Y 124.114,Z 420.325,A -85,B 0,C 180,E1 -27396.205,E2 -27396.205} C_VEL
LIN {X 0,Y 119.001,Z 428.848,A -85,B 0,C 180,E1 -27398.508,E2 -27398.508} C_VEL
LIN {X 0,Y 114.037,Z 436.06,A -85,B 0,C 180,E1 -27400.979,E2 -27400.979} C_VEL
LIN {X 0,Y 109.367,Z 442.258,A -85,B 0,C 180,E1 -27403.703,E2 -27403.703} C_VEL
LIN {X 0,Y 104.001,Z 448.795,A -85,B 0,C 180,E1 -27407.487,E2 -27407.487} C_VEL
LIN {X 0,Y 100.073,Z 453.297,A -85,B 0,C 180,E1 -27410.798,E2 -27410.798} C_VEL
LIN {X 0,Y 94.756,Z 458.789,A -85,B 0,C 180,E1 -27416.202,E2 -27416.202} C_VEL
LIN {X 0,Y 90.388,Z 463.116,A -85,B 0,C 180,E1 -27422.191,E2 -27422.191} C_VEL
LIN {X 0,Y 88.004,Z 465.486,A -85,B 0,C 180,E1 -27426.466,E2 -27426.466} C_VEL
LIN {X 0,Y 86.236,Z 467.293,A -85,B 0,C 180,E1 -27430.975,E2 -27430.975} C_VEL
LIN {X 0,Y 84.146,Z 469.756,A -85,B 0,C 180,E1 -27440.384,E2 -27440.384} C_VEL
LIN {X 0,Y 83.796,Z 470.354,A -85,B 0,C 180,E1 -27445.189,E2 -27445.189} C_VEL
LIN {X 0,Y 83.883,Z 470.516,A -85,B 0,C 180,E1 -27450,E2 -27450} C_VEL
LIN {X 0,Y 83.789,Z 470.353,A -85,B 0,C 180,E1 -27454.811,E2 -27454.811} C_VEL
LIN {X 0,Y 84.125,Z 469.755,A -85,B 0,C 180,E1 -27459.618,E2 -27459.618} C_VEL
LIN {X 0,Y 86.217,Z 467.292,A -85,B 0,C 180,E1 -27469.03,E2 -27469.03} C_VEL
LIN {X 0,Y 89.132,Z 464.334,A -85,B 0,C 180,E1 -27475.701,E2 -27475.701} C_VEL
LIN {X 0,Y 93.18,Z 460.343,A -85,B 0,C 180,E1 -27481.868,E2 -27481.868} C_VEL
LIN {X 0,Y 98.246,Z 455.214,A -85,B 0,C 180,E1 -27487.448,E2 -27487.448} C_VEL
LIN {X 0,Y 102.549,Z 450.469,A -85,B 0,C 180,E1 -27491.339,E2 -27491.339} C_VEL
LIN {X 0,Y 107.146,Z 445.009,A -85,B 0,C 180,E1 -27494.839,E2 -27494.839} C_VEL
LIN {X 0,Y 111.693,Z 439.313,A -85,B 0,C 180,E1 -27497.675,E2 -27497.675} C_VEL
LIN {X 0,Y 117.714,Z 430.765,A -85,B 0,C 180,E1 -27500.909,E2 -27500.909} C_VEL
LIN {X 0,Y 122.804,Z 422.592,A -85,B 0,C 180,E1 -27503.245,E2 -27503.245} C_VEL
LIN {X 0,Y 127.414,Z 414.085,A -85,B 0,C 180,E1 -27505.133,E2 -27505.133} C_VEL
LIN {X 0,Y 131.504,Z 405.377,A -85,B 0,C 180,E1 -27506.62,E2 -27506.62} C_VEL
LIN {X 0,Y 135.352,Z 395.625,A -85,B 0,C 180,E1 -27507.887,E2 -27507.887} C_VEL
LIN {X 0,Y 138.171,Z 386.835,A -85,B 0,C 180,E1 -27508.777,E2 -27508.777} C_VEL
LIN {X 0,Y 140.738,Z 376.384,A -85,B 0,C 180,E1 -27509.58,E2 -27509.58} C_VEL
LIN {X 0,Y 142.547,Z 366.033,A -85,B 0,C 180,E1 -27510.119,E2 -27510.119} C_VEL
LIN {X 0,Y 144.439,Z 346.812,A -85,B 0,C 180,E1 -27510.883,E2 -27510.883} C_VEL
LIN {X 0,Y 141.488,Z 337.369,A -85,B 0,C 180,E1 -27514.138,E2 -27514.138} C_VEL
LIN {X 0,Y 139.518,Z 332.296,A -85,B 0,C 180,E1 -27516.473,E2 -27516.473} C_VEL
LIN {X 0,Y 136.342,Z 326.351,A -85,B 0,C 180,E1 -27520.618,E2 -27520.618} C_VEL
LIN {X 0,Y 133.899,Z 322.263,A -85,B 0,C 180,E1 -27524.589,E2 -27524.589} C_VEL
LIN {X 0,Y 132.068,Z 318.879,A -85,B 0,C 180,E1 -27528.613,E2 -27528.613} C_VEL
LIN {X 0,Y 129.999,Z 314.336,A -85,B 0,C 180,E1 -27538.449,E2 -27538.449} C_VEL
LIN {X 0,Y 129.964,Z 314.189,A -85,B 0,C 180,E1 -27540.773,E2 -27540.773} C_VEL
LIN {X 0,Y 130.107,Z 314.927,A -85,B 0,C 180,E1 -27543.676,E2 -27543.676} C_VEL
LIN {X 0,Y 131.863,Z 318.66,A -85,B 0,C 180,E1 -27551.264,E2 -27551.264} C_VEL
LIN {X 0,Y 132.245,Z 319.17,A -85,B 0,C 180,E1 -27552.212,E2 -27552.212} C_VEL
LIN {X 0,Y 133.085,Z 322.008,A -85,B 0,C 180,E1 -27554.429,E2 -27554.429} C_VEL
LIN {X 0,Y 134.423,Z 328.329,A -85,B 0,C 180,E1 -27557.664,E2 -27557.664} C_VEL
LIN {X 0,Y 136.489,Z 336.252,A -85,B 0,C 180,E1 -27561.396,E2 -27561.396} C_VEL
LIN {X 0,Y 137.477,Z 338.457,A -85,B 0,C 180,E1 -27562.729,E2 -27562.729} C_VEL
LIN {X 0,Y 140.556,Z 345.27,A -85,B 0,C 180,E1 -27566.367,E2 -27566.367} C_VEL
LIN {X 0,Y 143.663,Z 353.212,A -85,B 0,C 180,E1 -27569.588,E2 -27569.588} C_VEL
LIN {X 0,Y 145.828,Z 360.029,A -85,B 0,C 180,E1 -27571.809,E2 -27571.809} C_VEL
LIN {X 0,Y 147.918,Z 369.146,A -85,B 0,C 180,E1 -27574.346,E2 -27574.346} C_VEL
LIN {X 0,Y 149.664,Z 378.586,A -85,B 0,C 180,E1 -27577.033,E2 -27577.033} C_VEL
LIN {X 0,Y 151.521,Z 387.816,A -85,B 0,C 180,E1 -27580.015,E2 -27580.015} C_VEL
LIN {X 0,Y 153.672,Z 396.837,A -85,B 0,C 180,E1 -27583.313,E2 -27583.313} C_VEL
LIN {X 0,Y 156.561,Z 406.259,A -85,B 0,C 180,E1 -27587.227,E2 -27587.227} C_VEL
LIN {X 0,Y 160.135,Z 414.918,A -85,B 0,C 180,E1 -27591.278,E2 -27591.278} C_VEL
LIN {X 0,Y 164.497,Z 422.568,A -85,B 0,C 180,E1 -27595.285,E2 -27595.285} C_VEL
LIN {X 0,Y 170.094,Z 429.876,A -85,B 0,C 180,E1 -27599.511,E2 -27599.511} C_VEL
LIN {X 0,Y 177.768,Z 437.255,A -85,B 0,C 180,E1 -27604.222,E2 -27604.222} C_VEL
LIN {X 0,Y 184.711,Z 442.103,A -85,B 0,C 180,E1 -27607.636,E2 -27607.636} C_VEL
LIN {X 0,Y 193.112,Z 446.673,A -85,B 0,C 180,E1 -27611.122,E2 -27611.122} C_VEL
LIN {X 0,Y 203.871,Z 451.084,A -85,B 0,C 180,E1 -27614.843,E2 -27614.843} C_VEL
LIN {X 0,Y 217.475,Z 455.204,A -85,B 0,C 180,E1 -27618.82,E2 -27618.82} C_VEL
LIN {X 0,Y 227.384,Z 457.616,A -85,B 0,C 180,E1 -27621.508,E2 -27621.508} C_VEL
LIN {X 0,Y 233.548,Z 458.95,A -85,B 0,C 180,E1 -27623.229,E2 -27623.229} C_VEL
LIN {X 0,Y 239.787,Z 460.187,A -85,B 0,C 180,E1 -27625.203,E2 -27625.203} C_VEL
LIN {X 0,Y 243.471,Z 460.921,A -85,B 0,C 180,E1 -27626.69,E2 -27626.69} C_VEL
LIN {X 0,Y 246.799,Z 461.414,A -85,B 0,C 180,E1 -27628.368,E2 -27628.368} C_VEL
LIN {X 0,Y 248.643,Z 461.554,A -85,B 0,C 180,E1 -27630,E2 -27630} C_VEL
LIN {X 0,Y 246.795,Z 461.414,A -85,B 0,C 180,E1 -27631.632,E2 -27631.632} C_VEL
LIN {X 0,Y 243.465,Z 460.921,A -85,B 0,C 180,E1 -27633.31,E2 -27633.31} C_VEL
LIN {X 0,Y 239.033,Z 460.036,A -85,B 0,C 180,E1 -27635.06,E2 -27635.06} C_VEL
LIN {X 0,Y 233.004,Z 458.839,A -85,B 0,C 180,E1 -27636.93,E2 -27636.93} C_VEL
LIN {X 0,Y 225.592,Z 457.247,A -85,B 0,C 180,E1 -27638.961,E2 -27638.961} C_VEL
LIN {X 0,Y 215.36,Z 454.648,A -85,B 0,C 180,E1 -27641.765,E2 -27641.765} C_VEL
LIN {X 0,Y 200.329,Z 449.8,A -85,B 0,C 180,E1 -27646.299,E2 -27646.299} C_VEL
LIN {X 0,Y 188.05,Z 444.096,A -85,B 0,C 180,E1 -27650.884,E2 -27650.884} C_VEL
LIN {X 0,Y 178.746,Z 437.995,A -85,B 0,C 180,E1 -27655.271,E2 -27655.271} C_VEL
LIN {X 0,Y 171.671,Z 431.611,A -85,B 0,C 180,E1 -27659.424,E2 -27659.424} C_VEL
LIN {X 0,Y 165.66,Z 424.285,A -85,B 0,C 180,E1 -27663.753,E2 -27663.753} C_VEL
LIN {X 0,Y 161.264,Z 417.134,A -85,B 0,C 180,E1 -27667.599,E2 -27667.599} C_VEL
LIN {X 0,Y 158.1,Z 410.39,A -85,B 0,C 180,E1 -27670.916,E2 -27670.916} C_VEL
LIN {X 0,Y 155.015,Z 401.464,A -85,B 0,C 180,E1 -27674.812,E2 -27674.812} C_VEL
LIN {X 0,Y 152.723,Z 392.947,A -85,B 0,C 180,E1 -27678.144,E2 -27678.144} C_VEL
LIN {X 0,Y 150.629,Z 383.528,A -85,B 0,C 180,E1 -27681.42,E2 -27681.42} C_VEL
LIN {X 0,Y 148.559,Z 372.666,A -85,B 0,C 180,E1 -27684.688,E2 -27684.688} C_VEL
LIN {X 0,Y 146.402,Z 362.039,A -85,B 0,C 180,E1 -27687.62,E2 -27687.62} C_VEL
LIN {X 0,Y 144.165,Z 354.62,A -85,B 0,C 180,E1 -27689.922,E2 -27689.922} C_VEL
LIN {X 0,Y 141.182,Z 346.829,A -85,B 0,C 180,E1 -27692.948,E2 -27692.948} C_VEL
LIN {X 0,Y 138.456,Z 340.589,A -85,B 0,C 180,E1 -27696.043,E2 -27696.043} C_VEL
LIN {X 0,Y 135.552,Z 334.682,A -85,B 0,C 180,E1 -27699.888,E2 -27699.888} C_VEL
LIN {X 0,Y 133.762,Z 331.332,A -85,B 0,C 180,E1 -27702.713,E2 -27702.713} C_VEL
LIN {X 0,Y 132.53,Z 328.993,A -85,B 0,C 180,E1 -27705.02,E2 -27705.02} C_VEL
LIN {X 0,Y 130.826,Z 325.569,A -85,B 0,C 180,E1 -27709.129,E2 -27709.129} C_VEL
LIN {X 0,Y 129.26,Z 322.552,A -85,B 0,C 180,E1 -27715.714,E2 -27715.714} C_VEL
LIN {X 0,Y 129.113,Z 321.362,A -85,B 0,C 180,E1 -27718.442,E2 -27718.442} C_VEL
LIN {X 0,Y 129.109,Z 321.243,A -85,B 0,C 180,E1 -27720.781,E2 -27720.781} C_VEL
LIN {X 0,Y 129.24,Z 322.458,A -85,B 0,C 180,E1 -27723.704,E2 -27723.704} C_VEL
LIN {X 0,Y 131.033,Z 326.032,A -85,B 0,C 180,E1 -27731.086,E2 -27731.086} C_VEL
LIN {X 0,Y 133.252,Z 330.285,A -85,B 0,C 180,E1 -27735.979,E2 -27735.979} C_VEL
LIN {X 0,Y 135.473,Z 334.5,A -85,B 0,C 180,E1 -27739.61,E2 -27739.61} C_VEL
LIN {X 0,Y 137.792,Z 339.355,A -85,B 0,C 180,E1 -27742.778,E2 -27742.778} C_VEL
LIN {X 0,Y 139.864,Z 345.97,A -85,B 0,C 180,E1 -27745.484,E2 -27745.484} C_VEL
LIN {X 0,Y 140.843,Z 349.446,A -85,B 0,C 180,E1 -27746.687,E2 -27746.687} C_VEL
LIN {X 0,Y 138.729,Z 368.983,A -85,B 0,C 180,E1 -27747.478,E2 -27747.478} C_VEL
LIN {X 0,Y 135.723,Z 382.781,A -85,B 0,C 180,E1 -27748.323,E2 -27748.323} C_VEL
LIN {X 0,Y 132.457,Z 393.42,A -85,B 0,C 180,E1 -27749.29,E2 -27749.29} C_VEL
LIN {X 0,Y 128.458,Z 403.553,A -85,B 0,C 180,E1 -27750.494,E2 -27750.494} C_VEL
LIN {X 0,Y 124.191,Z 412.542,A -85,B 0,C 180,E1 -27751.913,E2 -27751.913} C_VEL
LIN {X 0,Y 119.375,Z 421.265,A -85,B 0,C 180,E1 -27753.738,E2 -27753.738} C_VEL
LIN {X 0,Y 114.702,Z 428.655,A -85,B 0,C 180,E1 -27755.723,E2 -27755.723} C_VEL
LIN {X 0,Y 109.515,Z 435.868,A -85,B 0,C 180,E1 -27758.175,E2 -27758.175} C_VEL
LIN {X 0,Y 104.58,Z 442.065,A -85,B 0,C 180,E1 -27760.885,E2 -27760.885} C_VEL
LIN {X 0,Y 98.857,Z 448.601,A -85,B 0,C 180,E1 -27764.69,E2 -27764.69} C_VEL
LIN {X 0,Y 94.65,Z 453.104,A -85,B 0,C 180,E1 -27768.067,E2 -27768.067} C_VEL
LIN {X 0,Y 88.929,Z 458.595,A -85,B 0,C 180,E1 -27773.65,E2 -27773.65} C_VEL
LIN {X 0,Y 84.144,Z 462.923,A -85,B 0,C 180,E1 -27779.925,E2 -27779.925} C_VEL
LIN {X 0,Y 81.51,Z 465.292,A -85,B 0,C 180,E1 -27784.462,E2 -27784.462} C_VEL
LIN {X 0,Y 79.52,Z 467.099,A -85,B 0,C 180,E1 -27789.297,E2 -27789.297} C_VEL
LIN {X 0,Y 77.131,Z 469.563,A -85,B 0,C 180,E1 -27799.5,E2 -27799.5} C_VEL
LIN {X 0,Y 76.733,Z 470.161,A -85,B 0,C 180,E1 -27804.745,E2 -27804.745} C_VEL
LIN {X 0,Y 76.781,Z 470.323,A -85,B 0,C 180,E1 -27810,E2 -27810} C_VEL
LIN {X 0,Y 76.709,Z 470.16,A -85,B 0,C 180,E1 -27815.257,E2 -27815.257} C_VEL
LIN {X 0,Y 77.113,Z 469.562,A -85,B 0,C 180,E1 -27820.502,E2 -27820.502} C_VEL
LIN {X 0,Y 79.504,Z 467.098,A -85,B 0,C 180,E1 -27830.707,E2 -27830.707} C_VEL
LIN {X 0,Y 82.767,Z 464.141,A -85,B 0,C 180,E1 -27837.841,E2 -27837.841} C_VEL
LIN {X 0,Y 87.196,Z 460.149,A -85,B 0,C 180,E1 -27844.347,E2 -27844.347} C_VEL
LIN {X 0,Y 92.679,Z 455.02,A -85,B 0,C 180,E1 -27850.133,E2 -27850.133} C_VEL
LIN {X 0,Y 97.772,Z 449.758,A -85,B 0,C 180,E1 -27854.493,E2 -27854.493} C_VEL
LIN {X 0,Y 103.374,Z 443.44,A -85,B 0,C 180,E1 -27858.404,E2 -27858.404} C_VEL
LIN {X 0,Y 108.254,Z 437.493,A -85,B 0,C 180,E1 -27861.174,E2 -27861.174} C_VEL
LIN {X 0,Y 113.364,Z 430.571,A -85,B 0,C 180,E1 -27863.7,E2 -27863.7} C_VEL
LIN {X 0,Y 118.684,Z 422.399,A -85,B 0,C 180,E1 -27865.998,E2 -27865.998} C_VEL
LIN {X 0,Y 123.497,Z 413.893,A -85,B 0,C 180,E1 -27867.834,E2 -27867.834} C_VEL
LIN {X 0,Y 127.745,Z 405.184,A -85,B 0,C 180,E1 -27869.274,E2 -27869.274} C_VEL
LIN {X 0,Y 131.714,Z 395.432,A -85,B 0,C 180,E1 -27870.505,E2 -27870.505} C_VEL
LIN {X 0,Y 134.63,Z 386.643,A -85,B 0,C 180,E1 -27871.36,E2 -27871.36} C_VEL
LIN {X 0,Y 137.302,Z 376.142,A -85,B 0,C 180,E1 -27872.131,E2 -27872.131} C_VEL
LIN {X 0,Y 139.141,Z 365.943,A -85,B 0,C 180,E1 -27872.644,E2 -27872.644} C_VEL
LIN {X 0,Y 140.846,Z 349.42,A -85,B 0,C 180,E1 -27873.313,E2 -27873.313} C_VEL
LIN {X 0,Y 138.41,Z 341.179,A -85,B 0,C 180,E1 -27876.394,E2 -27876.394} C_VEL
LIN {X 0,Y 137.19,Z 337.942,A -85,B 0,C 180,E1 -27878.014,E2 -27878.014} C_VEL
LIN {X 0,Y 134.6,Z 332.715,A -85,B 0,C 180,E1 -27881.741,E2 -27881.741} C_VEL
LIN {X 0,Y 132.436,Z 328.809,A -85,B 0,C 180,E1 -27885.595,E2 -27885.595} C_VEL
LIN {X 0,Y 130.779,Z 325.596,A -85,B 0,C 180,E1 -27889.612,E2 -27889.612} C_VEL
LIN {X 0,Y 129.13,Z 321.416,A -85,B 0,C 180,E1 -27898.439,E2 -27898.439} C_VEL
LIN {X 0,Y 129.097,Z 321.247,A -85,B 0,C 180,E1 -27900.778,E2 -27900.778} C_VEL
LIN {X 0,Y 129.189,Z 322,A -85,B 0,C 180,E1 -27903.312,E2 -27903.312} C_VEL
LIN {X 0,Y 131.087,Z 326.134,A -85,B 0,C 180,E1 -27911.614,E2 -27911.614} C_VEL
LIN {X 0,Y 133.353,Z 330.515,A -85,B 0,C 180,E1 -27916.552,E2 -27916.552} C_VEL
LIN {X 0,Y 135.21,Z 333.985,A -85,B 0,C 180,E1 -27919.6,E2 -27919.6} C_VEL
LIN {X 0,Y 137.477,Z 338.457,A -85,B 0,C 180,E1 -27922.729,E2 -27922.729} C_VEL
LIN {X 0,Y 138.455,Z 340.779,A -85,B 0,C 180,E1 -27923.975,E2 -27923.975} C_VEL
LIN {X 0,Y 139.58,Z 345.21,A -85,B 0,C 180,E1 -27925.519,E2 -27925.519} C_VEL
LIN {X 0,Y 140.374,Z 350.257,A -85,B 0,C 180,E1 -27926.78,E2 -27926.78} C_VEL
LIN {X 0,Y 141.76,Z 360.987,A -85,B 0,C 180,E1 -27929.138,E2 -27929.138} C_VEL
LIN {X 0,Y 142.375,Z 364.33,A -85,B 0,C 180,E1 -27930.048,E2 -27930.048} C_VEL
LIN {X 0,Y 144.142,Z 374.598,A -85,B 0,C 180,E1 -27933.071,E2 -27933.071} C_VEL
LIN {X 0,Y 145.929,Z 387.113,A -85,B 0,C 180,E1 -27937.05,E2 -27937.05} C_VEL
LIN {X 0,Y 147.728,Z 397.213,A -85,B 0,C 180,E1 -27940.852,E2 -27940.852} C_VEL
LIN {X 0,Y 149.829,Z 406.283,A -85,B 0,C 180,E1 -27944.714,E2 -27944.714} C_VEL
LIN {X 0,Y 152.677,Z 415.026,A -85,B 0,C 180,E1 -27948.937,E2 -27948.937} C_VEL
LIN {X 0,Y 156.406,Z 422.831,A -85,B 0,C 180,E1 -27953.205,E2 -27953.205} C_VEL
LIN {X 0,Y 161.252,Z 430.161,A -85,B 0,C 180,E1 -27957.648,E2 -27957.648} C_VEL
LIN {X 0,Y 167.185,Z 436.618,A -85,B 0,C 180,E1 -27961.976,E2 -27961.976} C_VEL
LIN {X 0,Y 174.39,Z 442.402,A -85,B 0,C 180,E1 -27966.234,E2 -27966.234} C_VEL
LIN {X 0,Y 181.365,Z 446.595,A -85,B 0,C 180,E1 -27969.589,E2 -27969.589} C_VEL
LIN {X 0,Y 190.745,Z 450.789,A -85,B 0,C 180,E1 -27973.325,E2 -27973.325} C_VEL
LIN {X 0,Y 205.766,Z 455.521,A -85,B 0,C 180,E1 -27978.175,E2 -27978.175} C_VEL
LIN {X 0,Y 214.308,Z 457.557,A -85,B 0,C 180,E1 -27980.563,E2 -27980.563} C_VEL
LIN {X 0,Y 222.38,Z 459.131,A -85,B 0,C 180,E1 -27982.738,E2 -27982.738} C_VEL
LIN {X 0,Y 229.36,Z 460.297,A -85,B 0,C 180,E1 -27984.726,E2 -27984.726} C_VEL
LIN {X 0,Y 232.571,Z 460.811,A -85,B 0,C 180,E1 -27985.709,E2 -27985.709} C_VEL
LIN {X 0,Y 234.919,Z 461.155,A -85,B 0,C 180,E1 -27986.57,E2 -27986.57} C_VEL
LIN {X 0,Y 239.044,Z 461.641,A -85,B 0,C 180,E1 -27988.372,E2 -27988.372} C_VEL
LIN {X 0,Y 241.287,Z 461.75,A -85,B 0,C 180,E1 -27990,E2 -27990} C_VEL
LIN {X 0,Y 238.921,Z 461.627,A -85,B 0,C 180,E1 -27991.686,E2 -27991.686} C_VEL
LIN {X 0,Y 234.917,Z 461.155,A -85,B 0,C 180,E1 -27993.43,E2 -27993.43} C_VEL
LIN {X 0,Y 232.571,Z 460.811,A -85,B 0,C 180,E1 -27994.291,E2 -27994.291} C_VEL
LIN {X 0,Y 226.212,Z 459.818,A -85,B 0,C 180,E1 -27996.194,E2 -27996.194} C_VEL
LIN {X 0,Y 219.952,Z 458.676,A -85,B 0,C 180,E1 -27997.902,E2 -27997.902} C_VEL
LIN {X 0,Y 207.793,Z 456.029,A -85,B 0,C 180,E1 -28001.24,E2 -28001.24} C_VEL
LIN {X 0,Y 196.225,Z 452.73,A -85,B 0,C 180,E1 -28004.758,E2 -28004.758} C_VEL
LIN {X 0,Y 185.458,Z 448.546,A -85,B 0,C 180,E1 -28008.673,E2 -28008.673} C_VEL
LIN {X 0,Y 178.048,Z 444.711,A -85,B 0,C 180,E1 -28011.94,E2 -28011.94} C_VEL
LIN {X 0,Y 171.286,Z 440.185,A -85,B 0,C 180,E1 -28015.491,E2 -28015.491} C_VEL
LIN {X 0,Y 163.41,Z 432.76,A -85,B 0,C 180,E1 -28020.667,E2 -28020.667} C_VEL
LIN {X 0,Y 157.792,Z 425.263,A -85,B 0,C 180,E1 -28025.381,E2 -28025.381} C_VEL
LIN {X 0,Y 153.621,Z 417.394,A -85,B 0,C 180,E1 -28029.828,E2 -28029.828} C_VEL
LIN {X 0,Y 151.301,Z 411.23,A -85,B 0,C 180,E1 -28032.983,E2 -28032.983} C_VEL
LIN {X 0,Y 148.465,Z 401.031,A -85,B 0,C 180,E1 -28037.598,E2 -28037.598} C_VEL
LIN {X 0,Y 146.785,Z 392.464,A -85,B 0,C 180,E1 -28041.002,E2 -28041.002} C_VEL
LIN {X 0,Y 145.204,Z 382.463,A -85,B 0,C 180,E1 -28044.495,E2 -28044.495} C_VEL
LIN {X 0,Y 143.73,Z 372.021,A -85,B 0,C 180,E1 -28047.671,E2 -28047.671} C_VEL
LIN {X 0,Y 142.088,Z 363.089,A -85,B 0,C 180,E1 -28050.357,E2 -28050.357} C_VEL
LIN {X 0,Y 139.799,Z 355.511,A -85,B 0,C 180,E1 -28053.101,E2 -28053.101} C_VEL
LIN {X 0,Y 136.924,Z 347.99,A -85,B 0,C 180,E1 -28056.562,E2 -28056.562} C_VEL
LIN {X 0,Y 134.173,Z 341.755,A -85,B 0,C 180,E1 -28060.431,E2 -28060.431} C_VEL
LIN {X 0,Y 132.19,Z 337.785,A -85,B 0,C 180,E1 -28063.794,E2 -28063.794} C_VEL
LIN {X 0,Y 131.037,Z 335.466,A -85,B 0,C 180,E1 -28066.174,E2 -28066.174} C_VEL
LIN {X 0,Y 129.73,Z 332.499,A -85,B 0,C 180,E1 -28069.682,E2 -28069.682} C_VEL
LIN {X 0,Y 128.29,Z 329.147,A -85,B 0,C 180,E1 -28076.861,E2 -28076.861} C_VEL
LIN {X 0,Y 128.233,Z 328.286,A -85,B 0,C 180,E1 -28079.217,E2 -28079.217} C_VEL
LIN {X 0,Y 128.248,Z 328.406,A -85,B 0,C 180,E1 -28081.179,E2 -28081.179} C_VEL
LIN {X 0,Y 129.884,Z 332.963,A -85,B 0,C 180,E1 -28090.448,E2 -28090.448} C_VEL
LIN {X 0,Y 131.806,Z 336.97,A -85,B 0,C 180,E1 -28095.068,E2 -28095.068} C_VEL
LIN {X 0,Y 133.553,Z 340.506,A -85,B 0,C 180,E1 -28098.209,E2 -28098.209} C_VEL
LIN {X 0,Y 135.534,Z 344.993,A -85,B 0,C 180,E1 -28101.226,E2 -28101.226} C_VEL
LIN {X 0,Y 137.354,Z 351.54,A -85,B 0,C 180,E1 -28103.92,E2 -28103.92} C_VEL
LIN {X 0,Y 137.51,Z 352.112,A -85,B 0,C 180,E1 -28104.136,E2 -28104.136} C_VEL
LIN {X 0,Y 135.428,Z 369.879,A -85,B 0,C 180,E1 -28104.86,E2 -28104.86} C_VEL
LIN {X 0,Y 132.506,Z 382.588,A -85,B 0,C 180,E1 -28105.623,E2 -28105.623} C_VEL
LIN {X 0,Y 129.136,Z 393.228,A -85,B 0,C 180,E1 -28106.546,E2 -28106.546} C_VEL
LIN {X 0,Y 125.012,Z 403.361,A -85,B 0,C 180,E1 -28107.694,E2 -28107.694} C_VEL
LIN {X 0,Y 120.584,Z 412.349,A -85,B 0,C 180,E1 -28109.045,E2 -28109.045} C_VEL
LIN {X 0,Y 115.584,Z 421.073,A -85,B 0,C 180,E1 -28110.811,E2 -28110.811} C_VEL
LIN {X 0,Y 110.703,Z 428.462,A -85,B 0,C 180,E1 -28112.736,E2 -28112.736} C_VEL
LIN {X 0,Y 105.261,Z 435.674,A -85,B 0,C 180,E1 -28115.125,E2 -28115.125} C_VEL
LIN {X 0,Y 100.058,Z 441.871,A -85,B 0,C 180,E1 -28117.797,E2 -28117.797} C_VEL
LIN {X 0,Y 93.973,Z 448.407,A -85,B 0,C 180,E1 -28121.594,E2 -28121.594} C_VEL
LIN {X 0,Y 88.379,Z 453.874,A -85,B 0,C 180,E1 -28125.92,E2 -28125.92} C_VEL
LIN {X 0,Y 83.305,Z 458.402,A -85,B 0,C 180,E1 -28130.748,E2 -28130.748} C_VEL
LIN {X 0,Y 78.057,Z 462.729,A -85,B 0,C 180,E1 -28137.302,E2 -28137.302} C_VEL
LIN {X 0,Y 75.137,Z 465.099,A -85,B 0,C 180,E1 -28142.116,E2 -28142.116} C_VEL
LIN {X 0,Y 72.892,Z 466.905,A -85,B 0,C 180,E1 -28147.315,E2 -28147.315} C_VEL
LIN {X 0,Y 70.15,Z 469.369,A -85,B 0,C 180,E1 -28158.441,E2 -28158.441} C_VEL
LIN {X 0,Y 69.645,Z 469.968,A -85,B 0,C 180,E1 -28164.208,E2 -28164.208} C_VEL
LIN {X 0,Y 69.677,Z 470.131,A -85,B 0,C 180,E1 -28170,E2 -28170} C_VEL
LIN {X 0,Y 69.621,Z 469.967,A -85,B 0,C 180,E1 -28175.794,E2 -28175.794} C_VEL
LIN {X 0,Y 70.112,Z 469.368,A -85,B 0,C 180,E1 -28181.565,E2 -28181.565} C_VEL
LIN {X 0,Y 72.879,Z 466.905,A -85,B 0,C 180,E1 -28192.689,E2 -28192.689} C_VEL
LIN {X 0,Y 76.54,Z 463.947,A -85,B 0,C 180,E1 -28200.332,E2 -28200.332} C_VEL
LIN {X 0,Y 81.403,Z 459.955,A -85,B 0,C 180,E1 -28207.182,E2 -28207.182} C_VEL
LIN {X 0,Y 86.82,Z 455.315,A -85,B 0,C 180,E1 -28212.668,E2 -28212.668} C_VEL
LIN {X 0,Y 92.815,Z 449.564,A -85,B 0,C 180,E1 -28217.583,E2 -28217.583} C_VEL
LIN {X 0,Y 98.796,Z 443.247,A -85,B 0,C 180,E1 -28221.49,E2 -28221.49} C_VEL
LIN {X 0,Y 103.94,Z 437.3,A -85,B 0,C 180,E1 -28224.232,E2 -28224.232} C_VEL
LIN {X 0,Y 109.295,Z 430.378,A -85,B 0,C 180,E1 -28226.713,E2 -28226.713} C_VEL
LIN {X 0,Y 114.86,Z 422.206,A -85,B 0,C 180,E1 -28228.939,E2 -28228.939} C_VEL
LIN {X 0,Y 119.871,Z 413.7,A -85,B 0,C 180,E1 -28230.705,E2 -28230.705} C_VEL
LIN {X 0,Y 124.275,Z 404.992,A -85,B 0,C 180,E1 -28232.082,E2 -28232.082} C_VEL
LIN {X 0,Y 128.365,Z 395.24,A -85,B 0,C 180,E1 -28233.266,E2 -28233.266} C_VEL
LIN {X 0,Y 131.374,Z 386.45,A -85,B 0,C 180,E1 -28234.08,E2 -28234.08} C_VEL
LIN {X 0,Y 134.12,Z 376.031,A -85,B 0,C 180,E1 -28234.801,E2 -28234.801} C_VEL
LIN {X 0,Y 135.996,Z 366,A -85,B 0,C 180,E1 -28235.285,E2 -28235.285} C_VEL
LIN {X 0,Y 137.507,Z 352.142,A -85,B 0,C 180,E1 -28235.864,E2 -28235.864} C_VEL
LIN {X 0,Y 135.691,Z 345.424,A -85,B 0,C 180,E1 -28238.545,E2 -28238.545} C_VEL
LIN {X 0,Y 133.816,Z 341.03,A -85,B 0,C 180,E1 -28241.37,E2 -28241.37} C_VEL
LIN {X 0,Y 131.367,Z 335.95,A -85,B 0,C 180,E1 -28245.87,E2 -28245.87} C_VEL
LIN {X 0,Y 129.653,Z 332.46,A -85,B 0,C 180,E1 -28250.267,E2 -28250.267} C_VEL
LIN {X 0,Y 128.239,Z 328.333,A -85,B 0,C 180,E1 -28259.213,E2 -28259.213} C_VEL
LIN {X 0,Y 128.246,Z 328.423,A -85,B 0,C 180,E1 -28261.568,E2 -28261.568} C_VEL
LIN {X 0,Y 129.925,Z 333.044,A -85,B 0,C 180,E1 -28270.947,E2 -28270.947} C_VEL
LIN {X 0,Y 131.811,Z 336.984,A -85,B 0,C 180,E1 -28275.46,E2 -28275.46} C_VEL
LIN {X 0,Y 133.865,Z 341.132,A -85,B 0,C 180,E1 -28279.09,E2 -28279.09} C_VEL
LIN {X 0,Y 136.572,Z 347.11,A -85,B 0,C 180,E1 -28282.976,E2 -28282.976} C_VEL
LIN {X 0,Y 139.572,Z 354.89,A -85,B 0,C 180,E1 -28286.643,E2 -28286.643} C_VEL
LIN {X 0,Y 141.985,Z 362.8,A -85,B 0,C 180,E1 -28289.565,E2 -28289.565} C_VEL
LIN {X 0,Y 142.375,Z 364.33,A -85,B 0,C 180,E1 -28290.048,E2 -28290.048} C_VEL
LIN {X 0,Y 142.689,Z 367.82,A -85,B 0,C 180,E1 -28290.805,E2 -28290.805} C_VEL
LIN {X 0,Y 141.871,Z 374.265,A -85,B 0,C 180,E1 -28291.547,E2 -28291.547} C_VEL
LIN {X 0,Y 140.725,Z 380.677,A -85,B 0,C 180,E1 -28292.33,E2 -28292.33} C_VEL
LIN {X 0,Y 140.594,Z 384.121,A -85,B 0,C 180,E1 -28293.152,E2 -28293.152} C_VEL
LIN {X 0,Y 141.883,Z 396.176,A -85,B 0,C 180,E1 -28297.577,E2 -28297.577} C_VEL
LIN {X 0,Y 143.36,Z 405.797,A -85,B 0,C 180,E1 -28301.744,E2 -28301.744} C_VEL
LIN {X 0,Y 145.6,Z 415.106,A -85,B 0,C 180,E1 -28306.386,E2 -28306.386} C_VEL
LIN {X 0,Y 148.599,Z 423.121,A -85,B 0,C 180,E1 -28310.93,E2 -28310.93} C_VEL
LIN {X 0,Y 152.922,Z 430.754,A -85,B 0,C 180,E1 -28315.814,E2 -28315.814} C_VEL
LIN {X 0,Y 157.635,Z 436.575,A -85,B 0,C 180,E1 -28319.93,E2 -28319.93} C_VEL
LIN {X 0,Y 164.451,Z 442.692,A -85,B 0,C 180,E1 -28324.7,E2 -28324.7} C_VEL
LIN {X 0,Y 172.835,Z 447.938,A -85,B 0,C 180,E1 -28329.265,E2 -28329.265} C_VEL
LIN {X 0,Y 183.088,Z 452.439,A -85,B 0,C 180,E1 -28333.663,E2 -28333.663} C_VEL
LIN {X 0,Y 194.32,Z 455.927,A -85,B 0,C 180,E1 -28337.551,E2 -28337.551} C_VEL
LIN {X 0,Y 206.321,Z 458.577,A -85,B 0,C 180,E1 -28341.048,E2 -28341.048} C_VEL
LIN {X 0,Y 212.541,Z 459.673,A -85,B 0,C 180,E1 -28342.738,E2 -28342.738} C_VEL
LIN {X 0,Y 219.058,Z 460.574,A -85,B 0,C 180,E1 -28344.477,E2 -28344.477} C_VEL
LIN {X 0,Y 225.806,Z 461.404,A -85,B 0,C 180,E1 -28346.431,E2 -28346.431} C_VEL
LIN {X 0,Y 231.967,Z 461.927,A -85,B 0,C 180,E1 -28348.835,E2 -28348.835} C_VEL
LIN {X 0,Y 233.808,Z 461.949,A -85,B 0,C 180,E1 -28350,E2 -28350} C_VEL
LIN {X 0,Y 231.967,Z 461.927,A -85,B 0,C 180,E1 -28351.164,E2 -28351.164} C_VEL
LIN {X 0,Y 225.805,Z 461.404,A -85,B 0,C 180,E1 -28353.569,E2 -28353.569} C_VEL
LIN {X 0,Y 218.894,Z 460.557,A -85,B 0,C 180,E1 -28355.561,E2 -28355.561} C_VEL
LIN {X 0,Y 206.317,Z 458.582,A -85,B 0,C 180,E1 -28358.946,E2 -28358.946} C_VEL
LIN {X 0,Y 193.972,Z 455.842,A -85,B 0,C 180,E1 -28362.556,E2 -28362.556} C_VEL
LIN {X 0,Y 180.42,Z 451.472,A -85,B 0,C 180,E1 -28367.385,E2 -28367.385} C_VEL
LIN {X 0,Y 168.148,Z 445.27,A -85,B 0,C 180,E1 -28373.148,E2 -28373.148} C_VEL
LIN {X 0,Y 159.797,Z 438.776,A -85,B 0,C 180,E1 -28378.407,E2 -28378.407} C_VEL
LIN {X 0,Y 153.904,Z 432.161,A -85,B 0,C 180,E1 -28383.228,E2 -28383.228} C_VEL
LIN {X 0,Y 149.774,Z 425.528,A -85,B 0,C 180,E1 -28387.59,E2 -28387.59} C_VEL
LIN {X 0,Y 146.985,Z 419.37,A -85,B 0,C 180,E1 -28391.303,E2 -28391.303} C_VEL
LIN {X 0,Y 144.347,Z 410.286,A -85,B 0,C 180,E1 -28396.07,E2 -28396.07} C_VEL
LIN {X 0,Y 142.637,Z 401.439,A -85,B 0,C 180,E1 -28400.17,E2 -28400.17} C_VEL
LIN {X 0,Y 141.54,Z 393.602,A -85,B 0,C 180,E1 -28403.429,E2 -28403.429} C_VEL
LIN {X 0,Y 140.513,Z 383.263,A -85,B 0,C 180,E1 -28407.122,E2 -28407.122} C_VEL
LIN {X 0,Y 139.512,Z 372.919,A -85,B 0,C 180,E1 -28410.378,E2 -28410.378} C_VEL
LIN {X 0,Y 138.13,Z 364.7,A -85,B 0,C 180,E1 -28413.158,E2 -28413.158} C_VEL
LIN {X 0,Y 135.834,Z 356.884,A -85,B 0,C 180,E1 -28416.463,E2 -28416.463} C_VEL
LIN {X 0,Y 133.471,Z 350.622,A -85,B 0,C 180,E1 -28419.887,E2 -28419.887} C_VEL
LIN {X 0,Y 131.188,Z 345.256,A -85,B 0,C 180,E1 -28423.867,E2 -28423.867} C_VEL
LIN {X 0,Y 129.629,Z 341.963,A -85,B 0,C 180,E1 -28427.29,E2 -28427.29} C_VEL
LIN {X 0,Y 128.427,Z 339.128,A -85,B 0,C 180,E1 -28430.95,E2 -28430.95} C_VEL
LIN {X 0,Y 127.365,Z 335.35,A -85,B 0,C 180,E1 -28439.211,E2 -28439.211} C_VEL
LIN {X 0,Y 127.369,Z 335.569,A -85,B 0,C 180,E1 -28441.187,E2 -28441.187} C_VEL
LIN {X 0,Y 128.769,Z 339.902,A -85,B 0,C 180,E1 -28449.843,E2 -28449.843} C_VEL
LIN {X 0,Y 130.356,Z 343.519,A -85,B 0,C 180,E1 -28454.041,E2 -28454.041} C_VEL
LIN {X 0,Y 131.925,Z 346.998,A -85,B 0,C 180,E1 -28457.15,E2 -28457.15} C_VEL
LIN {X 0,Y 133.452,Z 350.847,A -85,B 0,C 180,E1 -28459.744,E2 -28459.744} C_VEL
LIN {X 0,Y 134.446,Z 354.919,A -85,B 0,C 180,E1 -28461.466,E2 -28461.466} C_VEL
LIN {X 0,Y 132.449,Z 370.418,A -85,B 0,C 180,E1 -28462.102,E2 -28462.102} C_VEL
LIN {X 0,Y 129.595,Z 382.396,A -85,B 0,C 180,E1 -28462.792,E2 -28462.792} C_VEL
LIN {X 0,Y 126.463,Z 392.151,A -85,B 0,C 180,E1 -28463.575,E2 -28463.575} C_VEL
LIN {X 0,Y 122.651,Z 401.538,A -85,B 0,C 180,E1 -28464.543,E2 -28464.543} C_VEL
LIN {X 0,Y 118.061,Z 410.806,A -85,B 0,C 180,E1 -28465.794,E2 -28465.794} C_VEL
LIN {X 0,Y 112.842,Z 419.746,A -85,B 0,C 180,E1 -28467.438,E2 -28467.438} C_VEL
LIN {X 0,Y 107.029,Z 428.269,A -85,B 0,C 180,E1 -28469.536,E2 -28469.536} C_VEL
LIN {X 0,Y 101.337,Z 435.481,A -85,B 0,C 180,E1 -28471.835,E2 -28471.835} C_VEL
LIN {X 0,Y 95.865,Z 441.678,A -85,B 0,C 180,E1 -28474.437,E2 -28474.437} C_VEL
LIN {X 0,Y 89.389,Z 448.213,A -85,B 0,C 180,E1 -28478.166,E2 -28478.166} C_VEL
LIN {X 0,Y 82.765,Z 454.208,A -85,B 0,C 180,E1 -28483.015,E2 -28483.015} C_VEL
LIN {X 0,Y 77.928,Z 458.209,A -85,B 0,C 180,E1 -28487.438,E2 -28487.438} C_VEL
LIN {X 0,Y 72.166,Z 462.536,A -85,B 0,C 180,E1 -28494.245,E2 -28494.245} C_VEL
LIN {X 0,Y 68.919,Z 464.905,A -85,B 0,C 180,E1 -28499.345,E2 -28499.345} C_VEL
LIN {X 0,Y 64.452,Z 468.108,A -85,B 0,C 180,E1 -28510.906,E2 -28510.906} C_VEL
LIN {X 0,Y 63.184,Z 469.176,A -85,B 0,C 180,E1 -28517.146,E2 -28517.146} C_VEL
LIN {X 0,Y 62.575,Z 469.775,A -85,B 0,C 180,E1 -28523.551,E2 -28523.551} C_VEL
LIN {X 0,Y 62.568,Z 469.938,A -85,B 0,C 180,E1 -28530,E2 -28530} C_VEL
LIN {X 0,Y 62.554,Z 469.774,A -85,B 0,C 180,E1 -28536.451,E2 -28536.451} C_VEL
LIN {X 0,Y 63.153,Z 469.175,A -85,B 0,C 180,E1 -28542.86,E2 -28542.86} C_VEL
LIN {X 0,Y 66.342,Z 466.711,A -85,B 0,C 180,E1 -28555.071,E2 -28555.071} C_VEL
LIN {X 0,Y 70.487,Z 463.754,A -85,B 0,C 180,E1 -28563.256,E2 -28563.256} C_VEL
LIN {X 0,Y 75.847,Z 459.762,A -85,B 0,C 180,E1 -28570.437,E2 -28570.437} C_VEL
LIN {X 0,Y 81.411,Z 455.386,A -85,B 0,C 180,E1 -28575.792,E2 -28575.792} C_VEL
LIN {X 0,Y 88.158,Z 449.369,A -85,B 0,C 180,E1 -28581.011,E2 -28581.011} C_VEL
LIN {X 0,Y 94.534,Z 443.054,A -85,B 0,C 180,E1 -28584.862,E2 -28584.862} C_VEL
LIN {X 0,Y 99.942,Z 437.107,A -85,B 0,C 180,E1 -28587.548,E2 -28587.548} C_VEL
LIN {X 0,Y 105.554,Z 430.185,A -85,B 0,C 180,E1 -28589.947,E2 -28589.947} C_VEL
LIN {X 0,Y 111.364,Z 422.013,A -85,B 0,C 180,E1 -28592.069,E2 -28592.069} C_VEL
LIN {X 0,Y 116.566,Z 413.508,A -85,B 0,C 180,E1 -28593.746,E2 -28593.746} C_VEL
LIN {X 0,Y 121.119,Z 404.8,A -85,B 0,C 180,E1 -28595.046,E2 -28595.046} C_VEL
LIN {X 0,Y 124.932,Z 396.115,A -85,B 0,C 180,E1 -28596.053,E2 -28596.053} C_VEL
LIN {X 0,Y 128.56,Z 385.836,A -85,B 0,C 180,E1 -28596.956,E2 -28596.956} C_VEL
LIN {X 0,Y 131.279,Z 375.687,A -85,B 0,C 180,E1 -28597.623,E2 -28597.623} C_VEL
LIN {X 0,Y 133.192,Z 365.807,A -85,B 0,C 180,E1 -28598.053,E2 -28598.053} C_VEL
LIN {X 0,Y 134.442,Z 354.958,A -85,B 0,C 180,E1 -28598.534,E2 -28598.534} C_VEL
LIN {X 0,Y 133.168,Z 349.946,A -85,B 0,C 180,E1 -28600.739,E2 -28600.739} C_VEL
LIN {X 0,Y 131.183,Z 345.229,A -85,B 0,C 180,E1 -28604.262,E2 -28604.262} C_VEL
LIN {X 0,Y 129.53,Z 341.747,A -85,B 0,C 180,E1 -28607.926,E2 -28607.926} C_VEL
LIN {X 0,Y 128.42,Z 339.155,A -85,B 0,C 180,E1 -28611.342,E2 -28611.342} C_VEL
LIN {X 0,Y 127.368,Z 335.368,A -85,B 0,C 180,E1 -28619.405,E2 -28619.405} C_VEL
LIN {X 0,Y 127.37,Z 335.655,A -85,B 0,C 180,E1 -28621.777,E2 -28621.777} C_VEL
LIN {X 0,Y 128.77,Z 339.865,A -85,B 0,C 180,E1 -28630.216,E2 -28630.216} C_VEL
LIN {X 0,Y 130.403,Z 343.653,A -85,B 0,C 180,E1 -28634.532,E2 -28634.532} C_VEL
LIN {X 0,Y 132.007,Z 347.195,A -85,B 0,C 180,E1 -28637.681,E2 -28637.681} C_VEL
LIN {X 0,Y 134.374,Z 352.851,A -85,B 0,C 180,E1 -28641.474,E2 -28641.474} C_VEL
LIN {X 0,Y 136.804,Z 360.015,A -85,B 0,C 180,E1 -28644.973,E2 -28644.973} C_VEL
LIN {X 0,Y 138.773,Z 367.745,A -85,B 0,C 180,E1 -28647.932,E2 -28647.932} C_VEL
LIN {X 0,Y 139.986,Z 377.142,A -85,B 0,C 180,E1 -28650.886,E2 -28650.886} C_VEL
LIN {X 0,Y 140.594,Z 384.121,A -85,B 0,C 180,E1 -28653.152,E2 -28653.152} C_VEL
LIN {X 0,Y 140.509,Z 387.497,A -85,B 0,C 180,E1 -28654.037,E2 -28654.037} C_VEL
LIN {X 0,Y 137.424,Z 399.47,A -85,B 0,C 180,E1 -28656.296,E2 -28656.296} C_VEL
LIN {X 0,Y 137.175,Z 402.534,A -85,B 0,C 180,E1 -28657.335,E2 -28657.335} C_VEL
LIN {X 0,Y 138.571,Z 412.777,A -85,B 0,C 180,E1 -28662.329,E2 -28662.329} C_VEL
LIN {X 0,Y 140.707,Z 421.813,A -85,B 0,C 180,E1 -28667.45,E2 -28667.45} C_VEL
LIN {X 0,Y 143.936,Z 429.583,A -85,B 0,C 180,E1 -28672.536,E2 -28672.536} C_VEL
LIN {X 0,Y 148.955,Z 437.101,A -85,B 0,C 180,E1 -28678.13,E2 -28678.13} C_VEL
LIN {X 0,Y 154.823,Z 442.977,A -85,B 0,C 180,E1 -28683.003,E2 -28683.003} C_VEL
LIN {X 0,Y 162.833,Z 448.487,A -85,B 0,C 180,E1 -28688.114,E2 -28688.114} C_VEL
LIN {X 0,Y 170.165,Z 452.073,A -85,B 0,C 180,E1 -28691.787,E2 -28691.787} C_VEL
LIN {X 0,Y 182.363,Z 456.159,A -85,B 0,C 180,E1 -28696.63,E2 -28696.63} C_VEL
LIN {X 0,Y 192.704,Z 458.564,A -85,B 0,C 180,E1 -28699.958,E2 -28699.958} C_VEL
LIN {X 0,Y 205.154,Z 460.549,A -85,B 0,C 180,E1 -28703.432,E2 -28703.432} C_VEL
LIN {X 0,Y 215.658,Z 461.682,A -85,B 0,C 180,E1 -28706.263,E2 -28706.263} C_VEL
LIN {X 0,Y 221.885,Z 462.088,A -85,B 0,C 180,E1 -28708.185,E2 -28708.185} C_VEL
LIN {X 0,Y 224.907,Z 462.168,A -85,B 0,C 180,E1 -28709.32,E2 -28709.32} C_VEL
LIN {X 0,Y 226.164,Z 462.153,A -85,B 0,C 180,E1 -28710,E2 -28710} C_VEL
LIN {X 0,Y 224.907,Z 462.168,A -85,B 0,C 180,E1 -28710.68,E2 -28710.68} C_VEL
LIN {X 0,Y 221.884,Z 462.088,A -85,B 0,C 180,E1 -28711.815,E2 -28711.815} C_VEL
LIN {X 0,Y 215.658,Z 461.682,A -85,B 0,C 180,E1 -28713.737,E2 -28713.737} C_VEL
LIN {X 0,Y 205.146,Z 460.561,A -85,B 0,C 180,E1 -28716.549,E2 -28716.549} C_VEL
LIN {X 0,Y 190.774,Z 458.206,A -85,B 0,C 180,E1 -28720.614,E2 -28720.614} C_VEL
LIN {X 0,Y 175.436,Z 454.05,A -85,B 0,C 180,E1 -28725.967,E2 -28725.967} C_VEL
LIN {X 0,Y 165.191,Z 449.765,A -85,B 0,C 180,E1 -28730.617,E2 -28730.617} C_VEL
LIN {X 0,Y 158.392,Z 445.735,A -85,B 0,C 180,E1 -28734.553,E2 -28734.553} C_VEL
LIN {X 0,Y 150.637,Z 439.006,A -85,B 0,C 180,E1 -28740.337,E2 -28740.337} C_VEL
LIN {X 0,Y 145.913,Z 432.931,A -85,B 0,C 180,E1 -28745.036,E2 -28745.036} C_VEL
LIN {X 0,Y 142.136,Z 425.794,A -85,B 0,C 180,E1 -28750,E2 -28750} C_VEL
LIN {X 0,Y 139.829,Z 418.91,A -85,B 0,C 180,E1 -28754.261,E2 -28754.261} C_VEL
LIN {X 0,Y 138.179,Z 410.97,A -85,B 0,C 180,E1 -28758.611,E2 -28758.611} C_VEL
LIN {X 0,Y 137.101,Z 401.849,A -85,B 0,C 180,E1 -28762.967,E2 -28762.967} C_VEL
LIN {X 0,Y 136.538,Z 393.264,A -85,B 0,C 180,E1 -28766.555,E2 -28766.555} C_VEL
LIN {X 0,Y 136.091,Z 383.245,A -85,B 0,C 180,E1 -28770.198,E2 -28770.198} C_VEL
LIN {X 0,Y 135.563,Z 374.093,A -85,B 0,C 180,E1 -28773.233,E2 -28773.233} C_VEL
LIN {X 0,Y 134.591,Z 367.27,A -85,B 0,C 180,E1 -28775.823,E2 -28775.823} C_VEL
LIN {X 0,Y 132.59,Z 359.72,A -85,B 0,C 180,E1 -28779.443,E2 -28779.443} C_VEL
LIN {X 0,Y 130.438,Z 353.703,A -85,B 0,C 180,E1 -28783.369,E2 -28783.369} C_VEL
LIN {X 0,Y 128.545,Z 349.004,A -85,B 0,C 180,E1 -28787.693,E2 -28787.693} C_VEL
LIN {X 0,Y 127.445,Z 346.124,A -85,B 0,C 180,E1 -28791.279,E2 -28791.279} C_VEL
LIN {X 0,Y 126.504,Z 342.311,A -85,B 0,C 180,E1 -28799.841,E2 -28799.841} C_VEL
LIN {X 0,Y 127.586,Z 346.594,A -85,B 0,C 180,E1 -28808.914,E2 -28808.914} C_VEL
LIN {X 0,Y 129.168,Z 350.567,A -85,B 0,C 180,E1 -28813.515,E2 -28813.515} C_VEL
LIN {X 0,Y 130.764,Z 354.61,A -85,B 0,C 180,E1 -28816.893,E2 -28816.893} C_VEL
LIN {X 0,Y 131.492,Z 356.99,A -85,B 0,C 180,E1 -28818.303,E2 -28818.303} C_VEL
LIN {X 0,Y 131.68,Z 357.788,A -85,B 0,C 180,E1 -28818.679,E2 -28818.679} C_VEL
LIN {X 0,Y 129.857,Z 370.615,A -85,B 0,C 180,E1 -28819.218,E2 -28819.218} C_VEL
LIN {X 0,Y 127.019,Z 382.203,A -85,B 0,C 180,E1 -28819.845,E2 -28819.845} C_VEL
LIN {X 0,Y 123.616,Z 392.42,A -85,B 0,C 180,E1 -28820.607,E2 -28820.607} C_VEL
LIN {X 0,Y 119.881,Z 401.346,A -85,B 0,C 180,E1 -28821.461,E2 -28821.461} C_VEL
LIN {X 0,Y 115.147,Z 410.614,A -85,B 0,C 180,E1 -28822.608,E2 -28822.608} C_VEL
LIN {X 0,Y 109.742,Z 419.552,A -85,B 0,C 180,E1 -28824.135,E2 -28824.135} C_VEL
LIN {X 0,Y 103.711,Z 428.076,A -85,B 0,C 180,E1 -28826.119,E2 -28826.119} C_VEL
LIN {X 0,Y 97.765,Z 435.288,A -85,B 0,C 180,E1 -28828.284,E2 -28828.284} C_VEL
LIN {X 0,Y 92.033,Z 441.485,A -85,B 0,C 180,E1 -28830.785,E2 -28830.785} C_VEL
LIN {X 0,Y 85.165,Z 448.019,A -85,B 0,C 180,E1 -28834.389,E2 -28834.389} C_VEL
LIN {X 0,Y 79.009,Z 453.303,A -85,B 0,C 180,E1 -28838.514,E2 -28838.514} C_VEL
LIN {X 0,Y 72.848,Z 458.016,A -85,B 0,C 180,E1 -28843.651,E2 -28843.651} C_VEL
LIN {X 0,Y 66.519,Z 462.343,A -85,B 0,C 180,E1 -28850.66,E2 -28850.66} C_VEL
LIN {X 0,Y 62.901,Z 464.712,A -85,B 0,C 180,E1 -28856.037,E2 -28856.037} C_VEL
LIN {X 0,Y 57.762,Z 467.915,A -85,B 0,C 180,E1 -28868.591,E2 -28868.591} C_VEL
LIN {X 0,Y 56.272,Z 468.983,A -85,B 0,C 180,E1 -28875.535,E2 -28875.535} C_VEL
LIN {X 0,Y 55.529,Z 469.582,A -85,B 0,C 180,E1 -28882.729,E2 -28882.729} C_VEL
LIN {X 0,Y 55.48,Z 469.745,A -85,B 0,C 180,E1 -28890,E2 -28890} C_VEL
LIN {X 0,Y 55.489,Z 469.581,A -85,B 0,C 180,E1 -28897.276,E2 -28897.276} C_VEL
LIN {X 0,Y 56.246,Z 468.982,A -85,B 0,C 180,E1 -28904.472,E2 -28904.472} C_VEL
LIN {X 0,Y 59.946,Z 466.517,A -85,B 0,C 180,E1 -28917.966,E2 -28917.966} C_VEL
LIN {X 0,Y 64.655,Z 463.561,A -85,B 0,C 180,E1 -28926.716,E2 -28926.716} C_VEL
LIN {X 0,Y 70.579,Z 459.568,A -85,B 0,C 180,E1 -28934.189,E2 -28934.189} C_VEL
LIN {X 0,Y 77.376,Z 454.553,A -85,B 0,C 180,E1 -28940.291,E2 -28940.291} C_VEL
LIN {X 0,Y 83.842,Z 449.175,A -85,B 0,C 180,E1 -28944.814,E2 -28944.814} C_VEL
LIN {X 0,Y 90.618,Z 442.86,A -85,B 0,C 180,E1 -28948.552,E2 -28948.552} C_VEL
LIN {X 0,Y 96.308,Z 436.913,A -85,B 0,C 180,E1 -28951.126,E2 -28951.126} C_VEL
LIN {X 0,Y 102.175,Z 429.991,A -85,B 0,C 180,E1 -28953.405,E2 -28953.405} C_VEL
LIN {X 0,Y 108.221,Z 421.82,A -85,B 0,C 180,E1 -28955.391,E2 -28955.391} C_VEL
LIN {X 0,Y 113.597,Z 413.315,A -85,B 0,C 180,E1 -28956.967,E2 -28956.967} C_VEL
LIN {X 0,Y 118.303,Z 404.607,A -85,B 0,C 180,E1 -28958.16,E2 -28958.16} C_VEL
LIN {X 0,Y 122.135,Z 396.154,A -85,B 0,C 180,E1 -28959.071,E2 -28959.071} C_VEL
LIN {X 0,Y 125.603,Z 386.777,A -85,B 0,C 180,E1 -28959.848,E2 -28959.848} C_VEL
LIN {X 0,Y 128.626,Z 376.005,A -85,B 0,C 180,E1 -28960.524,E2 -28960.524} C_VEL
LIN {X 0,Y 130.724,Z 365.464,A -85,B 0,C 180,E1 -28960.949,E2 -28960.949} C_VEL
LIN {X 0,Y 131.712,Z 357.916,A -85,B 0,C 180,E1 -28961.26,E2 -28961.26} C_VEL
LIN {X 0,Y 130.912,Z 355.013,A -85,B 0,C 180,E1 -28962.825,E2 -28962.825} C_VEL
LIN {X 0,Y 129.286,Z 350.885,A -85,B 0,C 180,E1 -28966.201,E2 -28966.201} C_VEL
LIN {X 0,Y 128.202,Z 348.253,A -85,B 0,C 180,E1 -28969.023,E2 -28969.023} C_VEL
LIN {X 0,Y 127.328,Z 346.008,A -85,B 0,C 180,E1 -28972.067,E2 -28972.067} C_VEL
LIN {X 0,Y 126.503,Z 342.321,A -85,B 0,C 180,E1 -28979.998,E2 -28979.998} C_VEL
LIN {X 0,Y 126.484,Z 343.227,A -85,B 0,C 180,E1 -28982.387,E2 -28982.387} C_VEL
LIN {X 0,Y 127.59,Z 346.602,A -85,B 0,C 180,E1 -28989.31,E2 -28989.31} C_VEL
LIN {X 0,Y 129.031,Z 350.306,A -85,B 0,C 180,E1 -28993.583,E2 -28993.583} C_VEL
LIN {X 0,Y 130.683,Z 354.303,A -85,B 0,C 180,E1 -28997.102,E2 -28997.102} C_VEL
LIN {X 0,Y 132.706,Z 360.248,A -85,B 0,C 180,E1 -29000.842,E2 -29000.842} C_VEL
LIN {X 0,Y 134.621,Z 367.547,A -85,B 0,C 180,E1 -29004.273,E2 -29004.273} C_VEL
LIN {X 0,Y 135.604,Z 374.347,A -85,B 0,C 180,E1 -29006.862,E2 -29006.862} C_VEL
LIN {X 0,Y 136.224,Z 385.596,A -85,B 0,C 180,E1 -29010.583,E2 -29010.583} C_VEL
LIN {X 0,Y 136.784,Z 397.909,A -85,B 0,C 180,E1 -29015.308,E2 -29015.308} C_VEL
LIN {X 0,Y 137.175,Z 402.534,A -85,B 0,C 180,E1 -29017.335,E2 -29017.335} C_VEL
LIN {X 0,Y 137.159,Z 406.832,A -85,B 0,C 180,E1 -29019.053,E2 -29019.053} C_VEL
LIN {X 0,Y 135.68,Z 414.421,A -85,B 0,C 180,E1 -29021.712,E2 -29021.712} C_VEL
LIN {X 0,Y 134.37,Z 421.441,A -85,B 0,C 180,E1 -29024.58,E2 -29024.58} C_VEL
LIN {X 0,Y 134.575,Z 424.869,A -85,B 0,C 180,E1 -29026.585,E2 -29026.585} C_VEL
LIN {X 0,Y 136.554,Z 430.514,A -85,B 0,C 180,E1 -29030.531,E2 -29030.531} C_VEL
LIN {X 0,Y 140.229,Z 437.157,A -85,B 0,C 180,E1 -29035.741,E2 -29035.741} C_VEL
LIN {X 0,Y 145.496,Z 443.258,A -85,B 0,C 180,E1 -29041.116,E2 -29041.116} C_VEL
LIN {X 0,Y 152.977,Z 448.939,A -85,B 0,C 180,E1 -29046.751,E2 -29046.751} C_VEL
LIN {X 0,Y 159.994,Z 452.608,A -85,B 0,C 180,E1 -29050.804,E2 -29050.804} C_VEL
LIN {X 0,Y 170.896,Z 456.474,A -85,B 0,C 180,E1 -29055.715,E2 -29055.715} C_VEL
LIN {X 0,Y 179.157,Z 458.552,A -85,B 0,C 180,E1 -29058.72,E2 -29058.72} C_VEL
LIN {X 0,Y 191.405,Z 460.636,A -85,B 0,C 180,E1 -29062.464,E2 -29062.464} C_VEL
LIN {X 0,Y 204.823,Z 461.979,A -85,B 0,C 180,E1 -29066.065,E2 -29066.065} C_VEL
LIN {X 0,Y 212.408,Z 462.344,A -85,B 0,C 180,E1 -29068.104,E2 -29068.104} C_VEL
LIN {X 0,Y 218.076,Z 462.368,A -85,B 0,C 180,E1 -29070,E2 -29070} C_VEL
LIN {X 0,Y 211.004,Z 462.28,A -85,B 0,C 180,E1 -29072.291,E2 -29072.291} C_VEL
LIN {X 0,Y 204.323,Z 461.94,A -85,B 0,C 180,E1 -29074.069,E2 -29074.069} C_VEL
LIN {X 0,Y 191.403,Z 460.638,A -85,B 0,C 180,E1 -29077.532,E2 -29077.532} C_VEL
LIN {X 0,Y 179.041,Z 458.53,A -85,B 0,C 180,E1 -29081.319,E2 -29081.319} C_VEL
LIN {X 0,Y 167.79,Z 455.576,A -85,B 0,C 180,E1 -29085.561,E2 -29085.561} C_VEL
LIN {X 0,Y 156.638,Z 451.042,A -85,B 0,C 180,E1 -29091.035,E2 -29091.035} C_VEL
LIN {X 0,Y 148.815,Z 446.093,A -85,B 0,C 180,E1 -29096.198,E2 -29096.198} C_VEL
LIN {X 0,Y 141.725,Z 439.166,A -85,B 0,C 180,E1 -29102.544,E2 -29102.544} C_VEL
LIN {X 0,Y 137.557,Z 432.701,A -85,B 0,C 180,E1 -29107.814,E2 -29107.814} C_VEL
LIN {X 0,Y 134.692,Z 425.399,A -85,B 0,C 180,E1 -29113.074,E2 -29113.074} C_VEL
LIN {X 0,Y 133.168,Z 418.161,A -85,B 0,C 180,E1 -29117.634,E2 -29117.634} C_VEL
LIN {X 0,Y 132.365,Z 410.935,A -85,B 0,C 180,E1 -29121.684,E2 -29121.684} C_VEL
LIN {X 0,Y 131.983,Z 402.306,A -85,B 0,C 180,E1 -29125.928,E2 -29125.928} C_VEL
LIN {X 0,Y 132.005,Z 393.618,A -85,B 0,C 180,E1 -29129.617,E2 -29129.617} C_VEL
LIN {X 0,Y 132.127,Z 383.652,A -85,B 0,C 180,E1 -29133.292,E2 -29133.292} C_VEL
LIN {X 0,Y 131.888,Z 374.869,A -85,B 0,C 180,E1 -29136.445,E2 -29136.445} C_VEL
LIN {X 0,Y 130.81,Z 367.743,A -85,B 0,C 180,E1 -29139.767,E2 -29139.767} C_VEL
LIN {X 0,Y 129.476,Z 362.31,A -85,B 0,C 180,E1 -29142.937,E2 -29142.937} C_VEL
LIN {X 0,Y 127.847,Z 357.3,A -85,B 0,C 180,E1 -29146.996,E2 -29146.996} C_VEL
LIN {X 0,Y 126.361,Z 352.996,A -85,B 0,C 180,E1 -29152.009,E2 -29152.009} C_VEL
LIN {X 0,Y 125.631,Z 349.426,A -85,B 0,C 180,E1 -29160.002,E2 -29160.002} C_VEL
LIN {X 0,Y 126.484,Z 353.469,A -85,B 0,C 180,E1 -29168.188,E2 -29168.188} C_VEL
LIN {X 0,Y 127.803,Z 357.191,A -85,B 0,C 180,E1 -29172.507,E2 -29172.507} C_VEL
LIN {X 0,Y 129.169,Z 361.16,A -85,B 0,C 180,E1 -29175.842,E2 -29175.842} C_VEL
LIN {X 0,Y 127.195,Z 372.61,A -85,B 0,C 180,E1 -29176.319,E2 -29176.319} C_VEL
LIN {X 0,Y 124.785,Z 382.01,A -85,B 0,C 180,E1 -29176.775,E2 -29176.775} C_VEL
LIN {X 0,Y 121.086,Z 392.766,A -85,B 0,C 180,E1 -29177.516,E2 -29177.516} C_VEL
LIN {X 0,Y 116.659,Z 402.784,A -85,B 0,C 180,E1 -29178.407,E2 -29178.407} C_VEL
LIN {X 0,Y 111.807,Z 411.771,A -85,B 0,C 180,E1 -29179.46,E2 -29179.46} C_VEL
LIN {X 0,Y 106.254,Z 420.494,A -85,B 0,C 180,E1 -29180.889,E2 -29180.889} C_VEL
LIN {X 0,Y 100.777,Z 427.883,A -85,B 0,C 180,E1 -29182.478,E2 -29182.478} C_VEL
LIN {X 0,Y 94.602,Z 435.095,A -85,B 0,C 180,E1 -29184.488,E2 -29184.488} C_VEL
LIN {X 0,Y 88.595,Z 441.292,A -85,B 0,C 180,E1 -29186.82,E2 -29186.82} C_VEL
LIN {X 0,Y 81.356,Z 447.826,A -85,B 0,C 180,E1 -29190.248,E2 -29190.248} C_VEL
LIN {X 0,Y 74.097,Z 453.598,A -85,B 0,C 180,E1 -29194.691,E2 -29194.691} C_VEL
LIN {X 0,Y 68.132,Z 457.823,A -85,B 0,C 180,E1 -29199.318,E2 -29199.318} C_VEL
LIN {X 0,Y 61.18,Z 462.149,A -85,B 0,C 180,E1 -29206.43,E2 -29206.43} C_VEL
LIN {X 0,Y 57.14,Z 464.519,A -85,B 0,C 180,E1 -29212.049,E2 -29212.049} C_VEL
LIN {X 0,Y 53.751,Z 466.323,A -85,B 0,C 180,E1 -29218.466,E2 -29218.466} C_VEL
LIN {X 0,Y 49.395,Z 468.789,A -85,B 0,C 180,E1 -29233.467,E2 -29233.467} C_VEL
LIN {X 0,Y 48.486,Z 469.389,A -85,B 0,C 180,E1 -29241.666,E2 -29241.666} C_VEL
LIN {X 0,Y 48.375,Z 469.552,A -85,B 0,C 180,E1 -29250,E2 -29250} C_VEL
LIN {X 0,Y 48.436,Z 469.388,A -85,B 0,C 180,E1 -29258.343,E2 -29258.343} C_VEL
LIN {X 0,Y 49.372,Z 468.789,A -85,B 0,C 180,E1 -29266.541,E2 -29266.541} C_VEL
LIN {X 0,Y 53.742,Z 466.323,A -85,B 0,C 180,E1 -29281.54,E2 -29281.54} C_VEL
LIN {X 0,Y 59.086,Z 463.367,A -85,B 0,C 180,E1 -29290.859,E2 -29290.859} C_VEL
LIN {X 0,Y 65.664,Z 459.375,A -85,B 0,C 180,E1 -29298.521,E2 -29298.521} C_VEL
LIN {X 0,Y 72.311,Z 454.88,A -85,B 0,C 180,E1 -29304.095,E2 -29304.095} C_VEL
LIN {X 0,Y 79.945,Z 448.981,A -85,B 0,C 180,E1 -29308.995,E2 -29308.995} C_VEL
LIN {X 0,Y 87.119,Z 442.667,A -85,B 0,C 180,E1 -29312.546,E2 -29312.546} C_VEL
LIN {X 0,Y 93.082,Z 436.72,A -85,B 0,C 180,E1 -29314.963,E2 -29314.963} C_VEL
LIN {X 0,Y 99.191,Z 429.798,A -85,B 0,C 180,E1 -29317.085,E2 -29317.085} C_VEL
LIN {X 0,Y 105.462,Z 421.628,A -85,B 0,C 180,E1 -29318.9,E2 -29318.9} C_VEL
LIN {X 0,Y 111.008,Z 413.122,A -85,B 0,C 180,E1 -29320.346,E2 -29320.346} C_VEL
LIN {X 0,Y 115.851,Z 404.415,A -85,B 0,C 180,E1 -29321.418,E2 -29321.418} C_VEL
LIN {X 0,Y 119.671,Z 396.231,A -85,B 0,C 180,E1 -29322.226,E2 -29322.226} C_VEL
LIN {X 0,Y 123.39,Z 386.419,A -85,B 0,C 180,E1 -29322.957,E2 -29322.957} C_VEL
LIN {X 0,Y 126.444,Z 375.782,A -85,B 0,C 180,E1 -29323.558,E2 -29323.558} C_VEL
LIN {X 0,Y 128.62,Z 365.054,A -85,B 0,C 180,E1 -29323.94,E2 -29323.94} C_VEL
LIN {X 0,Y 129.164,Z 361.276,A -85,B 0,C 180,E1 -29324.101,E2 -29324.101} C_VEL
LIN {X 0,Y 127.876,Z 357.392,A -85,B 0,C 180,E1 -29327.299,E2 -29327.299} C_VEL
LIN {X 0,Y 126.779,Z 354.422,A -85,B 0,C 180,E1 -29330.626,E2 -29330.626} C_VEL
LIN {X 0,Y 126.257,Z 352.858,A -85,B 0,C 180,E1 -29332.803,E2 -29332.803} C_VEL
LIN {X 0,Y 125.63,Z 349.436,A -85,B 0,C 180,E1 -29339.998,E2 -29339.998} C_VEL
LIN {X 0,Y 126.485,Z 353.507,A -85,B 0,C 180,E1 -29348.586,E2 -29348.586} C_VEL
LIN {X 0,Y 127.735,Z 357.025,A -85,B 0,C 180,E1 -29352.712,E2 -29352.712} C_VEL
LIN {X 0,Y 128.943,Z 360.697,A -85,B 0,C 180,E1 -29355.914,E2 -29355.914} C_VEL
LIN {X 0,Y 130.549,Z 366.421,A -85,B 0,C 180,E1 -29359.557,E2 -29359.557} C_VEL
LIN {X 0,Y 131.68,Z 373.553,A -85,B 0,C 180,E1 -29362.97,E2 -29362.97} C_VEL
LIN {X 0,Y 132.109,Z 379.29,A -85,B 0,C 180,E1 -29365.186,E2 -29365.186} C_VEL
LIN {X 0,Y 132.062,Z 389.007,A -85,B 0,C 180,E1 -29368.615,E2 -29368.615} C_VEL
LIN {X 0,Y 131.935,Z 399.486,A -85,B 0,C 180,E1 -29372.814,E2 -29372.814} C_VEL
LIN {X 0,Y 132.184,Z 407.824,A -85,B 0,C 180,E1 -29376.735,E2 -29376.735} C_VEL
LIN {X 0,Y 132.876,Z 416.035,A -85,B 0,C 180,E1 -29381.125,E2 -29381.125} C_VEL
LIN {X 0,Y 134.26,Z 423.722,A -85,B 0,C 180,E1 -29385.812,E2 -29385.812} C_VEL
LIN {X 0,Y 134.575,Z 424.869,A -85,B 0,C 180,E1 -29386.585,E2 -29386.585} C_VEL
LIN {X 0,Y 134.993,Z 428.348,A -85,B 0,C 180,E1 -29388.642,E2 -29388.642} C_VEL
LIN {X 0,Y 134.356,Z 434.321,A -85,B 0,C 180,E1 -29392.031,E2 -29392.031} C_VEL
LIN {X 0,Y 134.234,Z 439.672,A -85,B 0,C 180,E1 -29395.537,E2 -29395.537} C_VEL
LIN {X 0,Y 135.382,Z 442.243,A -85,B 0,C 180,E1 -29397.713,E2 -29397.713} C_VEL
LIN {X 0,Y 141.305,Z 447.914,A -85,B 0,C 180,E1 -29403.538,E2 -29403.538} C_VEL
LIN {X 0,Y 149.925,Z 453.082,A -85,B 0,C 180,E1 -29409.637,E2 -29409.637} C_VEL
LIN {X 0,Y 160.145,Z 456.916,A -85,B 0,C 180,E1 -29414.895,E2 -29414.895} C_VEL
LIN {X 0,Y 171.597,Z 459.648,A -85,B 0,C 180,E1 -29419.398,E2 -29419.398} C_VEL
LIN {X 0,Y 184.554,Z 461.502,A -85,B 0,C 180,E1 -29423.44,E2 -29423.44} C_VEL
LIN {X 0,Y 197.09,Z 462.443,A -85,B 0,C 180,E1 -29426.782,E2 -29426.782} C_VEL
LIN {X 0,Y 203.874,Z 462.681,A -85,B 0,C 180,E1 -29428.542,E2 -29428.542} C_VEL
LIN {X 0,Y 208.904,Z 462.612,A -85,B 0,C 180,E1 -29430,E2 -29430} C_VEL
LIN {X 0,Y 201.79,Z 462.631,A -85,B 0,C 180,E1 -29431.996,E2 -29431.996} C_VEL
LIN {X 0,Y 190.459,Z 462.091,A -85,B 0,C 180,E1 -29434.939,E2 -29434.939} C_VEL
LIN {X 0,Y 175.79,Z 460.395,A -85,B 0,C 180,E1 -29439.202,E2 -29439.202} C_VEL
LIN {X 0,Y 165.74,Z 458.459,A -85,B 0,C 180,E1 -29442.771,E2 -29442.771} C_VEL
LIN {X 0,Y 152.643,Z 454.283,A -85,B 0,C 180,E1 -29448.802,E2 -29448.802} C_VEL
LIN {X 0,Y 145.411,Z 450.65,A -85,B 0,C 180,E1 -29453.324,E2 -29453.324} C_VEL
LIN {X 0,Y 139.314,Z 446.311,A -85,B 0,C 180,E1 -29458.185,E2 -29458.185} C_VEL
LIN {X 0,Y 134.55,Z 441.187,A -85,B 0,C 180,E1 -29463.311,E2 -29463.311} C_VEL
LIN {X 0,Y 130.299,Z 433.828,A -85,B 0,C 180,E1 -29469.776,E2 -29469.776} C_VEL
LIN {X 0,Y 128.331,Z 427.619,A -85,B 0,C 180,E1 -29474.61,E2 -29474.61} C_VEL
LIN {X 0,Y 127.315,Z 420.104,A -85,B 0,C 180,E1 -29479.656,E2 -29479.656} C_VEL
LIN {X 0,Y 127.036,Z 411.84,A -85,B 0,C 180,E1 -29484.491,E2 -29484.491} C_VEL
LIN {X 0,Y 127.274,Z 404.012,A -85,B 0,C 180,E1 -29488.497,E2 -29488.497} C_VEL
LIN {X 0,Y 127.91,Z 394.032,A -85,B 0,C 180,E1 -29492.828,E2 -29492.828} C_VEL
LIN {X 0,Y 128.574,Z 383.185,A -85,B 0,C 180,E1 -29496.908,E2 -29496.908} C_VEL
LIN {X 0,Y 128.605,Z 377.995,A -85,B 0,C 180,E1 -29499.028,E2 -29499.028} C_VEL
LIN {X 0,Y 127.844,Z 371.152,A -85,B 0,C 180,E1 -29502.506,E2 -29502.506} C_VEL
LIN {X 0,Y 126.915,Z 366.162,A -85,B 0,C 180,E1 -29505.981,E2 -29505.981} C_VEL
LIN {X 0,Y 125.875,Z 362.206,A -85,B 0,C 180,E1 -29509.75,E2 -29509.75} C_VEL
LIN {X 0,Y 125.176,Z 359.666,A -85,B 0,C 180,E1 -29513.15,E2 -29513.15} C_VEL
LIN {X 0,Y 124.738,Z 356.701,A -85,B 0,C 180,E1 -29520.002,E2 -29520.002} C_VEL
LIN {X 0,Y 125.335,Z 360.16,A -85,B 0,C 180,E1 -29527.25,E2 -29527.25} C_VEL
LIN {X 0,Y 126.383,Z 363.912,A -85,B 0,C 180,E1 -29531.631,E2 -29531.631} C_VEL
LIN {X 0,Y 126.762,Z 365.347,A -85,B 0,C 180,E1 -29532.926,E2 -29532.926} C_VEL
LIN {X 0,Y 124.056,Z 377.995,A -85,B 0,C 180,E1 -29533.418,E2 -29533.418} C_VEL
LIN {X 0,Y 120.187,Z 390.012,A -85,B 0,C 180,E1 -29534.054,E2 -29534.054} C_VEL
LIN {X 0,Y 115.443,Z 400.96,A -85,B 0,C 180,E1 -29534.884,E2 -29534.884} C_VEL
LIN {X 0,Y 110.471,Z 410.228,A -85,B 0,C 180,E1 -29535.799,E2 -29535.799} C_VEL
LIN {X 0,Y 104.736,Z 419.167,A -85,B 0,C 180,E1 -29537.02,E2 -29537.02} C_VEL
LIN {X 0,Y 98.273,Z 427.689,A -85,B 0,C 180,E1 -29538.635,E2 -29538.635} C_VEL
LIN {X 0,Y 91.886,Z 434.902,A -85,B 0,C 180,E1 -29540.455,E2 -29540.455} C_VEL
LIN {X 0,Y 85.61,Z 441.098,A -85,B 0,C 180,E1 -29542.55,E2 -29542.55} C_VEL
LIN {X 0,Y 78.001,Z 447.632,A -85,B 0,C 180,E1 -29545.709,E2 -29545.709} C_VEL
LIN {X 0,Y 72.158,Z 452.135,A -85,B 0,C 180,E1 -29548.768,E2 -29548.768} C_VEL
LIN {X 0,Y 63.848,Z 457.629,A -85,B 0,C 180,E1 -29554.356,E2 -29554.356} C_VEL
LIN {X 0,Y 56.223,Z 461.956,A -85,B 0,C 180,E1 -29561.408,E2 -29561.408} C_VEL
LIN {X 0,Y 51.716,Z 464.326,A -85,B 0,C 180,E1 -29567.197,E2 -29567.197} C_VEL
LIN {X 0,Y 47.811,Z 466.129,A -85,B 0,C 180,E1 -29573.986,E2 -29573.986} C_VEL
LIN {X 0,Y 42.612,Z 468.596,A -85,B 0,C 180,E1 -29590.74,E2 -29590.74} C_VEL
LIN {X 0,Y 41.458,Z 469.196,A -85,B 0,C 180,E1 -29600.24,E2 -29600.24} C_VEL
LIN {X 0,Y 41.286,Z 469.36,A -85,B 0,C 180,E1 -29610,E2 -29610} C_VEL
LIN {X 0,Y 41.417,Z 469.195,A -85,B 0,C 180,E1 -29619.77,E2 -29619.77} C_VEL
LIN {X 0,Y 42.592,Z 468.595,A -85,B 0,C 180,E1 -29629.27,E2 -29629.27} C_VEL
LIN {X 0,Y 47.804,Z 466.129,A -85,B 0,C 180,E1 -29646.02,E2 -29646.02} C_VEL
LIN {X 0,Y 53.895,Z 463.173,A -85,B 0,C 180,E1 -29655.825,E2 -29655.825} C_VEL
LIN {X 0,Y 61.186,Z 459.182,A -85,B 0,C 180,E1 -29663.517,E2 -29663.517} C_VEL
LIN {X 0,Y 69.605,Z 453.865,A -85,B 0,C 180,E1 -29669.675,E2 -29669.675} C_VEL
LIN {X 0,Y 76.515,Z 448.788,A -85,B 0,C 180,E1 -29673.578,E2 -29673.578} C_VEL
LIN {X 0,Y 84.078,Z 442.474,A -85,B 0,C 180,E1 -29676.849,E2 -29676.849} C_VEL
LIN {X 0,Y 90.303,Z 436.527,A -85,B 0,C 180,E1 -29679.054,E2 -29679.054} C_VEL
LIN {X 0,Y 96.642,Z 429.605,A -85,B 0,C 180,E1 -29680.976,E2 -29680.976} C_VEL
LIN {X 0,Y 103.117,Z 421.435,A -85,B 0,C 180,E1 -29682.587,E2 -29682.587} C_VEL
LIN {X 0,Y 108.823,Z 412.929,A -85,B 0,C 180,E1 -29683.874,E2 -29683.874} C_VEL
LIN {X 0,Y 113.789,Z 404.222,A -85,B 0,C 180,E1 -29684.807,E2 -29684.807} C_VEL
LIN {X 0,Y 118.217,Z 394.754,A -85,B 0,C 180,E1 -29685.63,E2 -29685.63} C_VEL
LIN {X 0,Y 121.866,Z 385.083,A -85,B 0,C 180,E1 -29686.226,E2 -29686.226} C_VEL
LIN {X 0,Y 124.798,Z 374.888,A -85,B 0,C 180,E1 -29686.699,E2 -29686.699} C_VEL
LIN {X 0,Y 126.736,Z 365.325,A -85,B 0,C 180,E1 -29687.071,E2 -29687.071} C_VEL
LIN {X 0,Y 125.625,Z 361.407,A -85,B 0,C 180,E1 -29691.148,E2 -29691.148} C_VEL
LIN {X 0,Y 125.112,Z 359.506,A -85,B 0,C 180,E1 -29693.952,E2 -29693.952} C_VEL
LIN {X 0,Y 124.738,Z 356.697,A -85,B 0,C 180,E1 -29699.998,E2 -29699.998} C_VEL
LIN {X 0,Y 125.283,Z 360.201,A -85,B 0,C 180,E1 -29707.654,E2 -29707.654} C_VEL
LIN {X 0,Y 126.174,Z 363.539,A -85,B 0,C 180,E1 -29711.647,E2 -29711.647} C_VEL
LIN {X 0,Y 127.328,Z 367.984,A -85,B 0,C 180,E1 -29715.403,E2 -29715.403} C_VEL
LIN {X 0,Y 128.095,Z 373.168,A -85,B 0,C 180,E1 -29718.595,E2 -29718.595} C_VEL
LIN {X 0,Y 128.594,Z 378.028,A -85,B 0,C 180,E1 -29720.974,E2 -29720.974} C_VEL
LIN {X 0,Y 128.553,Z 384.784,A -85,B 0,C 180,E1 -29723.695,E2 -29723.695} C_VEL
LIN {X 0,Y 127.731,Z 396.88,A -85,B 0,C 180,E1 -29728.316,E2 -29728.316} C_VEL
LIN {X 0,Y 127.105,Z 407.015,A -85,B 0,C 180,E1 -29732.97,E2 -29732.97} C_VEL
LIN {X 0,Y 127.031,Z 415.395,A -85,B 0,C 180,E1 -29737.484,E2 -29737.484} C_VEL
LIN {X 0,Y 127.713,Z 424.001,A -85,B 0,C 180,E1 -29742.898,E2 -29742.898} C_VEL
LIN {X 0,Y 129.378,Z 431.3,A -85,B 0,C 180,E1 -29748.213,E2 -29748.213} C_VEL
LIN {X 0,Y 131.947,Z 437.117,A -85,B 0,C 180,E1 -29753.028,E2 -29753.028} C_VEL
LIN {X 0,Y 135.382,Z 442.243,A -85,B 0,C 180,E1 -29757.713,E2 -29757.713} C_VEL
LIN {X 0,Y 136.729,Z 444.684,A -85,B 0,C 180,E1 -29759.919,E2 -29759.919} C_VEL
LIN {X 0,Y 138.948,Z 452.106,A -85,B 0,C 180,E1 -29766.626,E2 -29766.626} C_VEL
LIN {X 0,Y 140.84,Z 453.856,A -85,B 0,C 180,E1 -29768.775,E2 -29768.775} C_VEL
LIN {X 0,Y 141.751,Z 454.344,A -85,B 0,C 180,E1 -29769.445,E2 -29769.445} C_VEL
LIN {X 0,Y 148.727,Z 457.085,A -85,B 0,C 180,E1 -29773.529,E2 -29773.529} C_VEL
LIN {X 0,Y 158.149,Z 459.594,A -85,B 0,C 180,E1 -29777.86,E2 -29777.86} C_VEL
LIN {X 0,Y 172.591,Z 461.824,A -85,B 0,C 180,E1 -29782.983,E2 -29782.983} C_VEL
LIN {X 0,Y 183.173,Z 462.673,A -85,B 0,C 180,E1 -29785.986,E2 -29785.986} C_VEL
LIN {X 0,Y 190.576,Z 462.934,A -85,B 0,C 180,E1 -29787.887,E2 -29787.887} C_VEL
LIN {X 0,Y 198.95,Z 462.877,A -85,B 0,C 180,E1 -29790,E2 -29790} C_VEL
LIN {X 0,Y 189.901,Z 462.916,A -85,B 0,C 180,E1 -29792.273,E2 -29792.273} C_VEL
LIN {X 0,Y 176.608,Z 462.234,A -85,B 0,C 180,E1 -29795.826,E2 -29795.826} C_VEL
LIN {X 0,Y 164.066,Z 460.712,A -85,B 0,C 180,E1 -29799.866,E2 -29799.866} C_VEL
LIN {X 0,Y 152.514,Z 458.225,A -85,B 0,C 180,E1 -29804.609,E2 -29804.609} C_VEL
LIN {X 0,Y 144.703,Z 455.678,A -85,B 0,C 180,E1 -29808.728,E2 -29808.728} C_VEL
LIN {X 0,Y 135.886,Z 451.103,A -85,B 0,C 180,E1 -29814.914,E2 -29814.914} C_VEL
LIN {X 0,Y 130.293,Z 446.578,A -85,B 0,C 180,E1 -29820.344,E2 -29820.344} C_VEL
LIN {X 0,Y 125.49,Z 440.172,A -85,B 0,C 180,E1 -29827.058,E2 -29827.058} C_VEL
LIN {X 0,Y 123.203,Z 434.718,A -85,B 0,C 180,E1 -29832.137,E2 -29832.137} C_VEL
LIN {X 0,Y 121.93,Z 428.145,A -85,B 0,C 180,E1 -29837.477,E2 -29837.477} C_VEL
LIN {X 0,Y 121.595,Z 419.758,A -85,B 0,C 180,E1 -29843.316,E2 -29843.316} C_VEL
LIN {X 0,Y 122.112,Z 411.648,A -85,B 0,C 180,E1 -29848.127,E2 -29848.127} C_VEL
LIN {X 0,Y 123.083,Z 403.273,A -85,B 0,C 180,E1 -29852.374,E2 -29852.374} C_VEL
LIN {X 0,Y 124.393,Z 393.231,A -85,B 0,C 180,E1 -29856.706,E2 -29856.706} C_VEL
LIN {X 0,Y 125.338,Z 384.972,A -85,B 0,C 180,E1 -29859.936,E2 -29859.936} C_VEL
LIN {X 0,Y 125.404,Z 379.073,A -85,B 0,C 180,E1 -29862.808,E2 -29862.808} C_VEL
LIN {X 0,Y 125.056,Z 374.411,A -85,B 0,C 180,E1 -29865.665,E2 -29865.665} C_VEL
LIN {X 0,Y 124.439,Z 370.008,A -85,B 0,C 180,E1 -29869.425,E2 -29869.425} C_VEL
LIN {X 0,Y 123.897,Z 366.551,A -85,B 0,C 180,E1 -29873.692,E2 -29873.692} C_VEL
LIN {X 0,Y 123.674,Z 363.892,A -85,B 0,C 180,E1 -29880.002,E2 -29880.002} C_VEL
LIN {X 0,Y 124.023,Z 367.141,A -85,B 0,C 180,E1 -29886.714,E2 -29886.714} C_VEL
LIN {X 0,Y 124.542,Z 369.704,A -85,B 0,C 180,E1 -29889.861,E2 -29889.861} C_VEL
LIN {X 0,Y 121.451,Z 381.625,A -85,B 0,C 180,E1 -29890.348,E2 -29890.348} C_VEL
LIN {X 0,Y 117.671,Z 392.198,A -85,B 0,C 180,E1 -29890.891,E2 -29890.891} C_VEL
LIN {X 0,Y 113.825,Z 400.767,A -85,B 0,C 180,E1 -29891.428,E2 -29891.428} C_VEL
LIN {X 0,Y 108.756,Z 410.036,A -85,B 0,C 180,E1 -29892.206,E2 -29892.206} C_VEL
LIN {X 0,Y 102.884,Z 418.974,A -85,B 0,C 180,E1 -29893.241,E2 -29893.241} C_VEL
LIN {X 0,Y 96.236,Z 427.496,A -85,B 0,C 180,E1 -29894.618,E2 -29894.618} C_VEL
LIN {X 0,Y 89.654,Z 434.709,A -85,B 0,C 180,E1 -29896.203,E2 -29896.203} C_VEL
LIN {X 0,Y 83.137,Z 440.904,A -85,B 0,C 180,E1 -29898.008,E2 -29898.008} C_VEL
LIN {X 0,Y 75.186,Z 447.439,A -85,B 0,C 180,E1 -29900.814,E2 -29900.814} C_VEL
LIN {X 0,Y 67.316,Z 453.016,A -85,B 0,C 180,E1 -29904.445,E2 -29904.445} C_VEL
LIN {X 0,Y 60.11,Z 457.435,A -85,B 0,C 180,E1 -29908.731,E2 -29908.731} C_VEL
LIN {X 0,Y 51.77,Z 461.761,A -85,B 0,C 180,E1 -29915.46,E2 -29915.46} C_VEL
LIN {X 0,Y 46.729,Z 464.132,A -85,B 0,C 180,E1 -29921.237,E2 -29921.237} C_VEL
LIN {X 0,Y 42.247,Z 465.936,A -85,B 0,C 180,E1 -29928.285,E2 -29928.285} C_VEL
LIN {X 0,Y 35.971,Z 468.403,A -85,B 0,C 180,E1 -29946.999,E2 -29946.999} C_VEL
LIN {X 0,Y 34.478,Z 469.003,A -85,B 0,C 180,E1 -29958.238,E2 -29958.238} C_VEL
LIN {X 0,Y 34.174,Z 469.167,A -85,B 0,C 180,E1 -29970,E2 -29970} C_VEL
LIN {X 0,Y 34.42,Z 469.001,A -85,B 0,C 180,E1 -29981.782,E2 -29981.782} C_VEL
LIN {X 0,Y 35.953,Z 468.402,A -85,B 0,C 180,E1 -29993.014,E2 -29993.014} C_VEL
LIN {X 0,Y 42.24,Z 465.935,A -85,B 0,C 180,E1 -30011.722,E2 -30011.722} C_VEL
LIN {X 0,Y 49.194,Z 462.98,A -85,B 0,C 180,E1 -30021.789,E2 -30021.789} C_VEL
LIN {X 0,Y 57.243,Z 458.989,A -85,B 0,C 180,E1 -30029.251,E2 -30029.251} C_VEL
LIN {X 0,Y 65.547,Z 454.146,A -85,B 0,C 180,E1 -30034.6,E2 -30034.6} C_VEL
LIN {X 0,Y 73.619,Z 448.594,A -85,B 0,C 180,E1 -30038.556,E2 -30038.556} C_VEL
LIN {X 0,Y 81.544,Z 442.281,A -85,B 0,C 180,E1 -30041.45,E2 -30041.45} C_VEL
LIN {X 0,Y 88.014,Z 436.334,A -85,B 0,C 180,E1 -30043.377,E2 -30043.377} C_VEL
LIN {X 0,Y 94.562,Z 429.412,A -85,B 0,C 180,E1 -30045.056,E2 -30045.056} C_VEL
LIN {X 0,Y 101.217,Z 421.242,A -85,B 0,C 180,E1 -30046.431,E2 -30046.431} C_VEL
LIN {X 0,Y 107.068,Z 412.736,A -85,B 0,C 180,E1 -30047.528,E2 -30047.528} C_VEL
LIN {X 0,Y 112.139,Z 404.029,A -85,B 0,C 180,E1 -30048.308,E2 -30048.308} C_VEL
LIN {X 0,Y 116.457,Z 395.042,A -85,B 0,C 180,E1 -30048.98,E2 -30048.98} C_VEL
LIN {X 0,Y 119.779,Z 386.713,A -85,B 0,C 180,E1 -30049.412,E2 -30049.412} C_VEL
LIN {X 0,Y 123.265,Z 375.081,A -85,B 0,C 180,E1 -30049.896,E2 -30049.896} C_VEL
LIN {X 0,Y 124.537,Z 369.717,A -85,B 0,C 180,E1 -30050.144,E2 -30050.144} C_VEL
LIN {X 0,Y 123.874,Z 366.472,A -85,B 0,C 180,E1 -30054.3,E2 -30054.3} C_VEL
LIN {X 0,Y 123.633,Z 363.884,A -85,B 0,C 180,E1 -30060.405,E2 -30060.405} C_VEL
LIN {X 0,Y 123.949,Z 367.036,A -85,B 0,C 180,E1 -30066.919,E2 -30066.919} C_VEL
LIN {X 0,Y 124.556,Z 370.671,A -85,B 0,C 180,E1 -30071.285,E2 -30071.285} C_VEL
LIN {X 0,Y 125.203,Z 375.6,A -85,B 0,C 180,E1 -30075.149,E2 -30075.149} C_VEL
LIN {X 0,Y 125.408,Z 379.998,A -85,B 0,C 180,E1 -30077.694,E2 -30077.694} C_VEL
LIN {X 0,Y 125.288,Z 385.988,A -85,B 0,C 180,E1 -30080.471,E2 -30080.471} C_VEL
LIN {X 0,Y 123.807,Z 397.87,A -85,B 0,C 180,E1 -30085.194,E2 -30085.194} C_VEL
LIN {X 0,Y 122.542,Z 407.431,A -85,B 0,C 180,E1 -30089.631,E2 -30089.631} C_VEL
LIN {X 0,Y 121.753,Z 416.427,A -85,B 0,C 180,E1 -30094.641,E2 -30094.641} C_VEL
LIN {X 0,Y 121.625,Z 423.892,A -85,B 0,C 180,E1 -30099.464,E2 -30099.464} C_VEL
LIN {X 0,Y 122.43,Z 431.579,A -85,B 0,C 180,E1 -30105.251,E2 -30105.251} C_VEL
LIN {X 0,Y 124.298,Z 437.721,A -85,B 0,C 180,E1 -30110.592,E2 -30110.592} C_VEL
LIN {X 0,Y 127.865,Z 443.814,A -85,B 0,C 180,E1 -30116.658,E2 -30116.658} C_VEL
LIN {X 0,Y 133.774,Z 449.612,A -85,B 0,C 180,E1 -30123.264,E2 -30123.264} C_VEL
LIN {X 0,Y 139.963,Z 453.478,A -85,B 0,C 180,E1 -30128.231,E2 -30128.231} C_VEL
LIN {X 0,Y 141.751,Z 454.344,A -85,B 0,C 180,E1 -30129.445,E2 -30129.445} C_VEL
LIN {X 0,Y 144.28,Z 455.96,A -85,B 0,C 180,E1 -30131.498,E2 -30131.498} C_VEL
LIN {X 0,Y 148.705,Z 459.458,A -85,B 0,C 180,E1 -30136.457,E2 -30136.457} C_VEL
LIN {X 0,Y 152.211,Z 460.852,A -85,B 0,C 180,E1 -30139.078,E2 -30139.078} C_VEL
LIN {X 0,Y 154.639,Z 461.361,A -85,B 0,C 180,E1 -30140.207,E2 -30140.207} C_VEL
LIN {X 0,Y 169.645,Z 462.933,A -85,B 0,C 180,E1 -30145.247,E2 -30145.247} C_VEL
LIN {X 0,Y 182.768,Z 463.284,A -85,B 0,C 180,E1 -30148.742,E2 -30148.742} C_VEL
LIN {X 0,Y 187.796,Z 463.174,A -85,B 0,C 180,E1 -30150,E2 -30150} C_VEL
LIN {X 0,Y 175.936,Z 463.162,A -85,B 0,C 180,E1 -30152.995,E2 -30152.995} C_VEL
LIN {X 0,Y 160.819,Z 462.141,A -85,B 0,C 180,E1 -30157.533,E2 -30157.533} C_VEL
LIN {X 0,Y 150.576,Z 460.641,A -85,B 0,C 180,E1 -30161.441,E2 -30161.441} C_VEL
LIN {X 0,Y 144.891,Z 459.47,A -85,B 0,C 180,E1 -30164.052,E2 -30164.052} C_VEL
LIN {X 0,Y 134.668,Z 456.077,A -85,B 0,C 180,E1 -30170.058,E2 -30170.058} C_VEL
LIN {X 0,Y 126.262,Z 451.294,A -85,B 0,C 180,E1 -30177.056,E2 -30177.056} C_VEL
LIN {X 0,Y 121.463,Z 446.682,A -85,B 0,C 180,E1 -30182.97,E2 -30182.97} C_VEL
LIN {X 0,Y 118.027,Z 441.11,A -85,B 0,C 180,E1 -30189.28,E2 -30189.28} C_VEL
LIN {X 0,Y 116.16,Z 434.407,A -85,B 0,C 180,E1 -30195.818,E2 -30195.818} C_VEL
LIN {X 0,Y 115.88,Z 426.814,A -85,B 0,C 180,E1 -30202.039,E2 -30202.039} C_VEL
LIN {X 0,Y 116.609,Z 418.898,A -85,B 0,C 180,E1 -30207.541,E2 -30207.541} C_VEL
LIN {X 0,Y 117.603,Z 412.494,A -85,B 0,C 180,E1 -30211.442,E2 -30211.442} C_VEL
LIN {X 0,Y 119.418,Z 403.219,A -85,B 0,C 180,E1 -30216.136,E2 -30216.136} C_VEL
LIN {X 0,Y 121.272,Z 393.854,A -85,B 0,C 180,E1 -30220.163,E2 -30220.163} C_VEL
LIN {X 0,Y 122.306,Z 387.558,A -85,B 0,C 180,E1 -30222.861,E2 -30222.861} C_VEL
LIN {X 0,Y 122.538,Z 382.074,A -85,B 0,C 180,E1 -30225.894,E2 -30225.894} C_VEL
LIN {X 0,Y 122.562,Z 378.629,A -85,B 0,C 180,E1 -30228.422,E2 -30228.422} C_VEL
LIN {X 0,Y 122.285,Z 375.115,A -85,B 0,C 180,E1 -30231.949,E2 -30231.949} C_VEL
LIN {X 0,Y 122.112,Z 373.002,A -85,B 0,C 180,E1 -30235.049,E2 -30235.049} C_VEL
LIN {X 0,Y 122.228,Z 371.015,A -85,B 0,C 180,E1 -30240.002,E2 -30240.002} C_VEL
LIN {X 0,Y 122.253,Z 373.715,A -85,B 0,C 180,E1 -30245.776,E2 -30245.776} C_VEL
LIN {X 0,Y 122.312,Z 374.464,A -85,B 0,C 180,E1 -30246.77,E2 -30246.77} C_VEL
LIN {X 0,Y 119.774,Z 383.242,A -85,B 0,C 180,E1 -30247.09,E2 -30247.09} C_VEL
LIN {X 0,Y 116.225,Z 392.745,A -85,B 0,C 180,E1 -30247.507,E2 -30247.507} C_VEL
LIN {X 0,Y 111.776,Z 402.206,A -85,B 0,C 180,E1 -30247.992,E2 -30247.992} C_VEL
LIN {X 0,Y 106.621,Z 411.193,A -85,B 0,C 180,E1 -30248.611,E2 -30248.611} C_VEL
LIN {X 0,Y 100.64,Z 419.915,A -85,B 0,C 180,E1 -30249.466,E2 -30249.466} C_VEL
LIN {X 0,Y 94.693,Z 427.303,A -85,B 0,C 180,E1 -30250.455,E2 -30250.455} C_VEL
LIN {X 0,Y 87.933,Z 434.516,A -85,B 0,C 180,E1 -30251.744,E2 -30251.744} C_VEL
LIN {X 0,Y 81.222,Z 440.711,A -85,B 0,C 180,E1 -30253.234,E2 -30253.234} C_VEL
LIN {X 0,Y 72.958,Z 447.245,A -85,B 0,C 180,E1 -30255.572,E2 -30255.572} C_VEL
LIN {X 0,Y 66.474,Z 451.747,A -85,B 0,C 180,E1 -30257.914,E2 -30257.914} C_VEL
LIN {X 0,Y 57.022,Z 457.241,A -85,B 0,C 180,E1 -30262.425,E2 -30262.425} C_VEL
LIN {X 0,Y 47.978,Z 461.567,A -85,B 0,C 180,E1 -30268.49,E2 -30268.49} C_VEL
LIN {X 0,Y 42.368,Z 463.939,A -85,B 0,C 180,E1 -30273.964,E2 -30273.964} C_VEL
LIN {X 0,Y 37.223,Z 465.742,A -85,B 0,C 180,E1 -30280.955,E2 -30280.955} C_VEL
LIN {X 0,Y 29.533,Z 468.209,A -85,B 0,C 180,E1 -30301.58,E2 -30301.58} C_VEL
LIN {X 0,Y 27.546,Z 468.81,A -85,B 0,C 180,E1 -30315.218,E2 -30315.218} C_VEL
LIN {X 0,Y 27.064,Z 468.974,A -85,B 0,C 180,E1 -30330,E2 -30330} C_VEL
LIN {X 0,Y 27.5,Z 468.809,A -85,B 0,C 180,E1 -30344.807,E2 -30344.807} C_VEL
LIN {X 0,Y 29.518,Z 468.208,A -85,B 0,C 180,E1 -30358.437,E2 -30358.437} C_VEL
LIN {X 0,Y 37.218,Z 465.742,A -85,B 0,C 180,E1 -30379.054,E2 -30379.054} C_VEL
LIN {X 0,Y 45.134,Z 462.786,A -85,B 0,C 180,E1 -30388.918,E2 -30388.918} C_VEL
LIN {X 0,Y 53.953,Z 458.796,A -85,B 0,C 180,E1 -30395.759,E2 -30395.759} C_VEL
LIN {X 0,Y 61.867,Z 454.523,A -85,B 0,C 180,E1 -30400.071,E2 -30400.071} C_VEL
LIN {X 0,Y 69.697,Z 449.556,A -85,B 0,C 180,E1 -30403.324,E2 -30403.324} C_VEL
LIN {X 0,Y 77.906,Z 443.463,A -85,B 0,C 180,E1 -30405.874,E2 -30405.874} C_VEL
LIN {X 0,Y 84.567,Z 437.766,A -85,B 0,C 180,E1 -30407.55,E2 -30407.55} C_VEL
LIN {X 0,Y 92.982,Z 429.218,A -85,B 0,C 180,E1 -30409.294,E2 -30409.294} C_VEL
LIN {X 0,Y 99.787,Z 421.048,A -85,B 0,C 180,E1 -30410.405,E2 -30410.405} C_VEL
LIN {X 0,Y 105.762,Z 412.543,A -85,B 0,C 180,E1 -30411.285,E2 -30411.285} C_VEL
LIN {X 0,Y 110.919,Z 403.837,A -85,B 0,C 180,E1 -30411.899,E2 -30411.899} C_VEL
LIN {X 0,Y 115.574,Z 394.24,A -85,B 0,C 180,E1 -30412.461,E2 -30412.461} C_VEL
LIN {X 0,Y 119.221,Z 384.885,A -85,B 0,C 180,E1 -30412.862,E2 -30412.862} C_VEL
LIN {X 0,Y 122.315,Z 374.45,A -85,B 0,C 180,E1 -30413.233,E2 -30413.233} C_VEL
LIN {X 0,Y 122.149,Z 372.826,A -85,B 0,C 180,E1 -30415.874,E2 -30415.874} C_VEL
LIN {X 0,Y 122.224,Z 371.03,A -85,B 0,C 180,E1 -30419.998,E2 -30419.998} C_VEL
LIN {X 0,Y 122.159,Z 373.588,A -85,B 0,C 180,E1 -30425.984,E2 -30425.984} C_VEL
LIN {X 0,Y 122.465,Z 376.767,A -85,B 0,C 180,E1 -30429.912,E2 -30429.912} C_VEL
LIN {X 0,Y 122.555,Z 380.818,A -85,B 0,C 180,E1 -30433.259,E2 -30433.259} C_VEL
LIN {X 0,Y 122.373,Z 386.673,A -85,B 0,C 180,E1 -30436.686,E2 -30436.686} C_VEL
LIN {X 0,Y 121.508,Z 392.483,A -85,B 0,C 180,E1 -30439.29,E2 -30439.29} C_VEL
LIN {X 0,Y 119.821,Z 401.044,A -85,B 0,C 180,E1 -30442.863,E2 -30442.863} C_VEL
LIN {X 0,Y 118.169,Z 409.311,A -85,B 0,C 180,E1 -30446.861,E2 -30446.861} C_VEL
LIN {X 0,Y 117.054,Z 415.724,A -85,B 0,C 180,E1 -30450.434,E2 -30450.434} C_VEL
LIN {X 0,Y 115.976,Z 424.557,A -85,B 0,C 180,E1 -30456.27,E2 -30456.27} C_VEL
LIN {X 0,Y 115.93,Z 431.654,A -85,B 0,C 180,E1 -30461.822,E2 -30461.822} C_VEL
LIN {X 0,Y 116.956,Z 437.985,A -85,B 0,C 180,E1 -30467.57,E2 -30467.57} C_VEL
LIN {X 0,Y 119.662,Z 444.084,A -85,B 0,C 180,E1 -30474.033,E2 -30474.033} C_VEL
LIN {X 0,Y 124.513,Z 449.828,A -85,B 0,C 180,E1 -30481.027,E2 -30481.027} C_VEL
LIN {X 0,Y 130.209,Z 453.817,A -85,B 0,C 180,E1 -30486.568,E2 -30486.568} C_VEL
LIN {X 0,Y 138.086,Z 457.381,A -85,B 0,C 180,E1 -30492.219,E2 -30492.219} C_VEL
LIN {X 0,Y 144.968,Z 459.478,A -85,B 0,C 180,E1 -30495.972,E2 -30495.972} C_VEL
LIN {X 0,Y 154.639,Z 461.361,A -85,B 0,C 180,E1 -30500.207,E2 -30500.207} C_VEL
LIN {X 0,Y 158.28,Z 462.048,A -85,B 0,C 180,E1 -30501.893,E2 -30501.893} C_VEL
LIN {X 0,Y 163.259,Z 463.07,A -85,B 0,C 180,E1 -30504.929,E2 -30504.929} C_VEL
LIN {X 0,Y 167.466,Z 463.49,A -85,B 0,C 180,E1 -30507.256,E2 -30507.256} C_VEL
LIN {X 0,Y 171.38,Z 463.601,A -85,B 0,C 180,E1 -30508.752,E2 -30508.752} C_VEL
LIN {X 0,Y 172.889,Z 463.546,A -85,B 0,C 180,E1 -30509.172,E2 -30509.172} C_VEL
LIN {X 0,Y 176.213,Z 463.483,A -85,B 0,C 180,E1 -30510,E2 -30510} C_VEL
LIN {X 0,Y 161.996,Z 463.408,A -85,B 0,C 180,E1 -30513.803,E2 -30513.803} C_VEL
LIN {X 0,Y 149.095,Z 462.443,A -85,B 0,C 180,E1 -30518.164,E2 -30518.164} C_VEL
LIN {X 0,Y 137.278,Z 460.508,A -85,B 0,C 180,E1 -30523.424,E2 -30523.424} C_VEL
LIN {X 0,Y 127.824,Z 457.67,A -85,B 0,C 180,E1 -30529.262,E2 -30529.262} C_VEL
LIN {X 0,Y 120.47,Z 454.064,A -85,B 0,C 180,E1 -30535.508,E2 -30535.508} C_VEL
LIN {X 0,Y 114.328,Z 448.607,A -85,B 0,C 180,E1 -30543.59,E2 -30543.59} C_VEL
LIN {X 0,Y 110.85,Z 441.949,A -85,B 0,C 180,E1 -30551.849,E2 -30551.849} C_VEL
LIN {X 0,Y 109.894,Z 434.93,A -85,B 0,C 180,E1 -30559.047,E2 -30559.047} C_VEL
LIN {X 0,Y 110.498,Z 427.062,A -85,B 0,C 180,E1 -30565.775,E2 -30565.775} C_VEL
LIN {X 0,Y 112.082,Z 419.14,A -85,B 0,C 180,E1 -30571.384,E2 -30571.384} C_VEL
LIN {X 0,Y 113.872,Z 412.099,A -85,B 0,C 180,E1 -30575.617,E2 -30575.617} C_VEL
LIN {X 0,Y 116.241,Z 403.433,A -85,B 0,C 180,E1 -30579.982,E2 -30579.982} C_VEL
LIN {X 0,Y 118.702,Z 393.884,A -85,B 0,C 180,E1 -30584.109,E2 -30584.109} C_VEL
LIN {X 0,Y 119.601,Z 388.82,A -85,B 0,C 180,E1 -30586.797,E2 -30586.797} C_VEL
LIN {X 0,Y 119.913,Z 385.714,A -85,B 0,C 180,E1 -30588.882,E2 -30588.882} C_VEL
LIN {X 0,Y 120.041,Z 382.682,A -85,B 0,C 180,E1 -30591.586,E2 -30591.586} C_VEL
LIN {X 0,Y 120.104,Z 380.699,A -85,B 0,C 180,E1 -30594.134,E2 -30594.134} C_VEL
LIN {X 0,Y 120.197,Z 379.332,A -85,B 0,C 180,E1 -30596.65,E2 -30596.65} C_VEL
LIN {X 0,Y 120.45,Z 378.053,A -85,B 0,C 180,E1 -30600.002,E2 -30600.002} C_VEL
LIN {X 0,Y 120.271,Z 379.495,A -85,B 0,C 180,E1 -30603.352,E2 -30603.352} C_VEL
LIN {X 0,Y 119.72,Z 381.24,A -85,B 0,C 180,E1 -30603.66,E2 -30603.66} C_VEL
LIN {X 0,Y 116.136,Z 391.103,A -85,B 0,C 180,E1 -30603.943,E2 -30603.943} C_VEL
LIN {X 0,Y 111.881,Z 400.382,A -85,B 0,C 180,E1 -30604.282,E2 -30604.282} C_VEL
LIN {X 0,Y 106.661,Z 409.65,A -85,B 0,C 180,E1 -30604.727,E2 -30604.727} C_VEL
LIN {X 0,Y 100.585,Z 418.588,A -85,B 0,C 180,E1 -30605.338,E2 -30605.338} C_VEL
LIN {X 0,Y 93.664,Z 427.111,A -85,B 0,C 180,E1 -30606.177,E2 -30606.177} C_VEL
LIN {X 0,Y 86.765,Z 434.323,A -85,B 0,C 180,E1 -30607.137,E2 -30607.137} C_VEL
LIN {X 0,Y 79.896,Z 440.519,A -85,B 0,C 180,E1 -30608.272,E2 -30608.272} C_VEL
LIN {X 0,Y 71.377,Z 447.052,A -85,B 0,C 180,E1 -30610.06,E2 -30610.06} C_VEL
LIN {X 0,Y 64.637,Z 451.553,A -85,B 0,C 180,E1 -30611.883,E2 -30611.883} C_VEL
LIN {X 0,Y 54.699,Z 457.048,A -85,B 0,C 180,E1 -30615.498,E2 -30615.498} C_VEL
LIN {X 0,Y 45.011,Z 461.373,A -85,B 0,C 180,E1 -30620.472,E2 -30620.472} C_VEL
LIN {X 0,Y 38.839,Z 463.745,A -85,B 0,C 180,E1 -30625.21,E2 -30625.21} C_VEL
LIN {X 0,Y 32.988,Z 465.548,A -85,B 0,C 180,E1 -30631.551,E2 -30631.551} C_VEL
LIN {X 0,Y 23.512,Z 468.015,A -85,B 0,C 180,E1 -30653.287,E2 -30653.287} C_VEL
LIN {X 0,Y 20.752,Z 468.617,A -85,B 0,C 180,E1 -30670.205,E2 -30670.205} C_VEL
LIN {X 0,Y 19.969,Z 468.781,A -85,B 0,C 180,E1 -30690,E2 -30690} C_VEL
LIN {X 0,Y 20.693,Z 468.615,A -85,B 0,C 180,E1 -30709.854,E2 -30709.854} C_VEL
LIN {X 0,Y 23.5,Z 468.015,A -85,B 0,C 180,E1 -30726.736,E2 -30726.736} C_VEL
LIN {X 0,Y 32.985,Z 465.548,A -85,B 0,C 180,E1 -30748.459,E2 -30748.459} C_VEL
LIN {X 0,Y 41.901,Z 462.593,A -85,B 0,C 180,E1 -30757.295,E2 -30757.295} C_VEL
LIN {X 0,Y 51.442,Z 458.603,A -85,B 0,C 180,E1 -30763.008,E2 -30763.008} C_VEL
LIN {X 0,Y 60.971,Z 453.662,A -85,B 0,C 180,E1 -30766.909,E2 -30766.909} C_VEL
LIN {X 0,Y 69.682,Z 448.207,A -85,B 0,C 180,E1 -30769.534,E2 -30769.534} C_VEL
LIN {X 0,Y 78.185,Z 441.894,A -85,B 0,C 180,E1 -30771.408,E2 -30771.408} C_VEL
LIN {X 0,Y 85.045,Z 435.948,A -85,B 0,C 180,E1 -30772.597,E2 -30772.597} C_VEL
LIN {X 0,Y 91.927,Z 429.026,A -85,B 0,C 180,E1 -30773.65,E2 -30773.65} C_VEL
LIN {X 0,Y 98.85,Z 420.855,A -85,B 0,C 180,E1 -30774.477,E2 -30774.477} C_VEL
LIN {X 0,Y 104.921,Z 412.35,A -85,B 0,C 180,E1 -30775.122,E2 -30775.122} C_VEL
LIN {X 0,Y 110.144,Z 403.644,A -85,B 0,C 180,E1 -30775.553,E2 -30775.553} C_VEL
LIN {X 0,Y 114.856,Z 394.053,A -85,B 0,C 180,E1 -30775.975,E2 -30775.975} C_VEL
LIN {X 0,Y 118.548,Z 384.692,A -85,B 0,C 180,E1 -30776.272,E2 -30776.272} C_VEL
LIN {X 0,Y 119.718,Z 381.24,A -85,B 0,C 180,E1 -30776.35,E2 -30776.35} C_VEL
LIN {X 0,Y 120.28,Z 379.467,A -85,B 0,C 180,E1 -30776.648,E2 -30776.648} C_VEL
LIN {X 0,Y 120.449,Z 378.057,A -85,B 0,C 180,E1 -30779.998,E2 -30779.998} C_VEL
LIN {X 0,Y 120.207,Z 379.303,A -85,B 0,C 180,E1 -30783.35,E2 -30783.35} C_VEL
LIN {X 0,Y 120.083,Z 381.289,A -85,B 0,C 180,E1 -30786.72,E2 -30786.72} C_VEL
LIN {X 0,Y 119.962,Z 384.501,A -85,B 0,C 180,E1 -30790.121,E2 -30790.121} C_VEL
LIN {X 0,Y 119.839,Z 387.089,A -85,B 0,C 180,E1 -30792.119,E2 -30792.119} C_VEL
LIN {X 0,Y 118.902,Z 392.868,A -85,B 0,C 180,E1 -30795.423,E2 -30795.423} C_VEL
LIN {X 0,Y 117.339,Z 399.385,A -85,B 0,C 180,E1 -30798.234,E2 -30798.234} C_VEL
